  MoveC 456 to (-171.94, 224.64, -10) mm, rotated rx 180 ry 0 rz 0.01 deg; joints [37.11, -45.165, 102.078, -138.154, 64.775, 160.021] to (-186.27, 223.92, -10) mm, rotated rx 180 ry 0 rz 0.01 deg; joints [36.765, -44.661, 101.03, -138.337, 64.242, 159.776]
  MoveL 457 to (-214.9, 224.22, -10) mm, rotated rx -180 ry 0 rz 0.01 deg; joints [36.141, -43.585, 98.793, -138.602, 63.141, 159.21]
  MoveC 458 to (-228.22, 225.49, -10) mm, rotated rx -180 ry 0 rz 0.01 deg; joints [35.891, -43.043, 97.666, -138.663, 62.606, 158.897] to (-241.07, 229.24, -10) mm, rotated rx -180 ry 0 rz 0.01 deg; joints [35.728, -42.444, 96.418, -138.608, 62.056, 158.493]
  MoveC 459 to (-253.06, 235.13, -10) mm, rotated rx -180 ry 0 rz 0.01 deg; joints [35.648, -41.812, 95.099, -138.448, 61.51, 158.018] to (-264.01, 242.79, -10) mm, rotated rx 180 ry 0 rz 0.01 deg; joints [35.642, -41.163, 93.745, -138.197, 60.981, 157.485]
  MoveC 460 to (-273.96, 253.08, -10) mm, rotated rx 180 ry 0 rz 0.01 deg; joints [35.733, -40.471, 92.297, -137.818, 60.457, 156.859] to (-281.3, 265.37, -10) mm, rotated rx -180 ry 0 rz 0.01 deg; joints [35.933, -39.816, 90.927, -137.333, 60.013, 156.197]
  MoveC 461 to (-284.47, 273.38, -10) mm, rotated rx -180 ry 0 rz 0.01 deg; joints [36.095, -39.451, 90.161, -137.006, 59.789, 155.796] to (-286.87, 281.66, -10) mm, rotated rx 180 ry 0 rz 0.01 deg; joints [36.278, -39.106, 89.437, -136.663, 59.592, 155.397]
  MoveC 462 to (-286.56, 286.16, -10) mm, rotated rx -180 ry 0 rz 0.01 deg; joints [36.411, -38.984, 89.179, -136.47, 59.552, 155.217] to (-283.74, 289.67, -10) mm, rotated rx 180 ry 0 rz 0.01 deg; joints [36.567, -38.995, 89.198, -136.31, 59.626, 155.138]
  MoveC 463 to (-280.78, 292.97, -10) mm, rotated rx -180 ry 0 rz 0.01 deg; joints [36.721, -39.019, 89.242, -136.159, 59.709, 155.072] to (-279.73, 297.28, -10) mm, rotated rx 180 ry 0 rz 0.01 deg; joints [36.863, -38.932, 89.056, -135.972, 59.701, 154.917]
  MoveC 464 to (-279.69, 299.8, -10) mm, rotated rx 180 ry 0 rz 0.01 deg; joints [36.934, -38.857, 88.897, -135.864, 59.672, 154.812] to (-279.52, 302.32, -10) mm, rotated rx -180 ry 0 rz 0.01 deg; joints [37.007, -38.787, 88.749, -135.756, 59.649, 154.71]
  MoveC 465 to (-280.39, 304.88, -10) mm, rotated rx 180 ry 0 rz 0.01 deg; joints [37.06, -38.672, 88.51, -135.651, 59.583, 154.581] to (-282.85, 305.96, -10) mm, rotated rx 180 ry 0 rz 0.01 deg; joints [37.038, -38.536, 88.227, -135.613, 59.469, 154.473]
  MoveL 466 to (-366.69, 305.96, -10) mm, rotated rx 180 ry 0 rz 0.01 deg; joints [35.359, -34.828, 80.603, -135.633, 55.88, 152.188]
  MoveC 467 to (-369.42, 304.83, -10) mm, rotated rx 180 ry 0 rz 0.01 deg; joints [35.276, -34.736, 80.417, -135.676, 55.772, 152.159] to (-370.55, 302.11, -10) mm, rotated rx -180 ry 0 rz 0.01 deg; joints [35.181, -34.772, 80.494, -135.797, 55.755, 152.251]
  MoveL 468 to (-370.54, 98.69, -10) mm, rotated rx 180 ry 0 rz 0.01 deg; joints [29.276, -40.424, 92.448, -144.823, 58.123, 160.617]
  MoveC 469 to (-369.42, 95.8, -10) mm, rotated rx 180 ry 0 rz 0.01 deg; joints [29.206, -40.54, 92.694, -144.946, 58.204, 160.746] to (-366.65, 94.41, -10) mm, rotated rx -180 ry 0 rz 0.01 deg; joints [29.211, -40.693, 93.013, -145, 58.342, 160.855]
  MoveC 470 to (-361.84, 93.97, -10) mm, rotated rx -180 ry 0 rz 0.01 deg; joints [29.281, -40.911, 93.465, -145.005, 58.558, 160.971] to (-357.03, 93.56, -10) mm, rotated rx 180 ry 0 rz 0.01 deg; joints [29.353, -41.128, 93.915, -145.008, 58.774, 161.086]
  MoveC 471 to (-352.24, 92.78, -10) mm, rotated rx 180 ry 0 rz 0.01 deg; joints [29.412, -41.351, 94.377, -145.026, 58.991, 161.212] to (-347.65, 91.24, -10) mm, rotated rx -180 ry 0 rz 0.01 deg; joints [29.445, -41.582, 94.859, -145.075, 59.207, 161.36]
  MoveC 472 to (-337.46, 86.07, -10) mm, rotated rx 180 ry 0 rz 0.01 deg; joints [29.463, -42.13, 96.004, -145.257, 59.704, 161.746] to (-328.09, 79.55, -10) mm, rotated rx 180 ry 0 rz 0.01 deg; joints [29.425, -42.669, 97.134, -145.493, 60.177, 162.156]
  MoveC 473 to (-319.86, 71.59, -10) mm, rotated rx 180 ry 0 rz 0.01 deg; joints [29.318, -43.186, 98.222, -145.792, 60.614, 162.585] to (-313.25, 62.25, -10) mm, rotated rx 180 ry 0 rz 0.01 deg; joints [29.137, -43.662, 99.228, -146.155, 60.996, 163.023]
  MoveL 474 to (-295.27, 31.05, -10) mm, rotated rx -180 ry 0 rz 0.01 deg; joints [28.438, -45.048, 102.174, -147.375, 62.088, 164.363]
  MoveC 475 to (-292.31, 25.1, -10) mm, rotated rx 180 ry 0 rz 0.01 deg; joints [28.294, -45.288, 102.686, -147.609, 62.275, 164.603] to (-290.1, 18.82, -10) mm, rotated rx -180 ry 0 rz 0.01 deg; joints [28.123, -45.503, 103.148, -147.862, 62.435, 164.839]
  MoveC 476 to (-288.58, 12.36, -10) mm, rotated rx -180 ry 0 rz 0.01 deg; joints [27.933, -45.694, 103.558, -148.128, 62.567, 165.067] to (-287.65, 5.78, -10) mm, rotated rx -180 ry 0 rz 0.01 deg; joints [27.728, -45.861, 103.921, -148.404, 62.676, 165.287]
  MoveC 477 to (-286.3, 3.07, -10) mm, rotated rx 180 ry 0 rz 0.01 deg; joints [27.66, -45.968, 104.149, -148.51, 62.761, 165.393] to (-283.47, 1.97, -10) mm, rotated rx 180 ry 0 rz 0.01 deg; joints [27.673, -46.101, 104.429, -148.535, 62.89, 165.473]
  MoveL 478 to (-110.06, 1.97, -10) mm, rotated rx 180 ry 0 rz 0.01 deg; joints [31.113, -52.422, 117.77, -146.55, 69.684, 168.087]
  MoveC 479 to (-107.23, 3.06, -10) mm, rotated rx -180 ry 0 rz 0.01 deg; joints [31.215, -52.496, 117.927, -146.461, 69.776, 168.098] to (-105.84, 5.75, -10) mm, rotated rx -180 ry 0 rz 0.01 deg; joints [31.345, -52.491, 117.909, -146.324, 69.796, 168.043]
  MoveC 480 to (-104.8, 12.53, -10) mm, rotated rx -180 ry 0 rz 0.01 deg; joints [31.615, -52.393, 117.685, -146.018, 69.754, 167.869] to (-103.19, 19.2, -10) mm, rotated rx -180 ry 0 rz 0.01 deg; joints [31.892, -52.315, 117.505, -145.709, 69.734, 167.705]
  MoveC 481 to (-100.9, 25.67, -10) mm, rotated rx 180 ry 0 rz 0.01 deg; joints [32.178, -52.262, 117.379, -145.399, 69.742, 167.556] to (-97.83, 31.82, -10) mm, rotated rx -180 ry 0 rz 0.01 deg; joints [32.468, -52.241, 117.321, -145.09, 69.781, 167.426]
  MoveL 482 to (-79.89, 62.85, -10) mm, rotated rx -180 ry 0 rz 0.01 deg; joints [33.989, -52.192, 117.153, -143.496, 70.059, 166.797]
  MoveC 483 to (-73.14, 72.29, -10) mm, rotated rx -180 ry 0 rz 0.01 deg; joints [34.481, -52.212, 117.176, -142.99, 70.187, 166.621] to (-64.7, 80.26, -10) mm, rotated rx -180 ry 0 rz 0.01 deg; joints [34.964, -52.315, 117.38, -142.516, 70.39, 166.513]
  MoveC 484 to (-55.07, 86.69, -10) mm, rotated rx -180 ry 0 rz 0.01 deg; joints [35.424, -52.487, 117.731, -142.083, 70.651, 166.468] to (-44.63, 91.7, -10) mm, rotated rx -180 ry 0 rz 0.01 deg; joints [35.858, -52.711, 118.2, -141.692, 70.955, 166.477]
  MoveC 485 to (-40.32, 93.04, -10) mm, rotated rx 180 ry 0 rz 0.01 deg; joints [36.014, -52.82, 118.428, -141.559, 71.088, 166.502] to (-35.85, 93.69, -10) mm, rotated rx -180 ry 0 rz 0.01 deg; joints [36.15, -52.947, 118.699, -141.45, 71.235, 166.55]
  MoveC 486 to (-31.35, 94.03, -10) mm, rotated rx 180 ry 0 rz 0.01 deg; joints [36.276, -53.082, 118.985, -141.353, 71.386, 166.607] to (-26.86, 94.42, -10) mm, rotated rx -180 ry 0 rz 0.01 deg; joints [36.404, -53.215, 119.269, -141.254, 71.536, 166.663]
  MoveC 487 to (-24.09, 95.8, -10) mm, rotated rx 180 ry 0 rz 0.01 deg; joints [36.524, -53.271, 119.387, -141.145, 71.614, 166.664] to (-22.97, 98.68, -10) mm, rotated rx 180 ry 0 rz 0.01 deg; joints [36.653, -53.242, 119.318, -141.005, 71.617, 166.595]
  MoveL 488 to (-22.97, 302.11, -10) mm, rotated rx -180 ry 0 rz 0.01 deg; joints [43.096, -48.06, 108.004, -133, 69.13, 159.892]
  MoveC 489 to (-24.1, 304.84, -10) mm, rotated rx 180 ry 0 rz 0.01 deg; joints [43.143, -47.946, 107.762, -132.917, 69.06, 159.773] to (-26.83, 305.97, -10) mm, rotated rx -180 ry 0 rz 0.01 deg; joints [43.103, -47.828, 107.512, -132.92, 68.955, 159.685]
  MoveL 490 to (-110.7, 305.97, -10) mm, rotated rx 180 ry 0 rz 0.01 deg; joints [40.945, -45.062, 101.736, -134.176, 66.057, 158.173]
  MoveC 491 to (-113.15, 304.87, -10) mm, rotated rx 180 ry 0 rz 0.01 deg; joints [40.853, -45.009, 101.629, -134.25, 65.983, 158.169] to (-113.97, 302.32, -10) mm, rotated rx -180 ry 0 rz 0.01 deg; joints [40.761, -45.055, 101.728, -134.361, 65.984, 158.249]
  MoveC 492 to (-113.72, 293.56, -10) mm, rotated rx -180 ry 0 rz 0.01 deg; joints [40.516, -45.317, 102.286, -134.701, 66.096, 158.583] to (-114.89, 284.87, -10) mm, rotated rx -180 ry 0 rz 0.01 deg; joints [40.237, -45.525, 102.732, -135.058, 66.157, 158.885]
  MoveC 493 to (-117.34, 276.46, -10) mm, rotated rx 180 ry 0 rz 0.01 deg; joints [39.933, -45.678, 103.064, -135.421, 66.168, 159.151] to (-120.94, 268.47, -10) mm, rotated rx 180 ry 0 rz 0.01 deg; joints [39.612, -45.777, 103.284, -135.783, 66.133, 159.377]
  MoveC 494 to (-124.45, 262.63, -10) mm, rotated rx -180 ry 0 rz 0.01 deg; joints [39.355, -45.818, 103.378, -136.06, 66.076, 159.526] to (-128.5, 257.15, -10) mm, rotated rx 180 ry 0 rz 0.01 deg; joints [39.096, -45.828, 103.408, -136.329, 65.994, 159.651]
  MoveC 495 to (-133.13, 252.15, -10) mm, rotated rx -180 ry 0 rz 0.01 deg; joints [38.837, -45.804, 103.366, -136.587, 65.885, 159.747] to (-138.35, 247.76, -10) mm, rotated rx 180 ry 0 rz 0.01 deg; joints [38.582, -45.741, 103.242, -136.828, 65.747, 159.811]
  MoveC 496 to (-143.45, 244.23, -10) mm, rotated rx -180 ry 0 rz 0.01 deg; joints [38.357, -45.657, 103.072, -137.032, 65.601, 159.844] to (-148.78, 241.05, -10) mm, rotated rx 180 ry 0 rz 0.01 deg; joints [38.137, -45.555, 102.864, -137.224, 65.443, 159.86]
  MoveC 497 to (-154.39, 238.38, -10) mm, rotated rx 180 ry 0 rz 0.01 deg; joints [37.926, -45.427, 102.603, -137.398, 65.267, 159.853] to (-160.28, 236.41, -10) mm, rotated rx 180 ry 0 rz 0.01 deg; joints [37.731, -45.27, 102.278, -137.546, 65.072, 159.814]
  MoveC 498 to (-173.77, 233.82, -10) mm, rotated rx 180 ry 0 rz 0.01 deg; joints [37.343, -44.853, 101.413, -137.802, 64.598, 159.654] to (-187.5, 233.2, -10) mm, rotated rx -180 ry 0 rz 0.01 deg; joints [37.015, -44.367, 100.404, -137.971, 64.087, 159.415]
  MoveL 499 to (-214.9, 233.58, -10) mm, rotated rx -180 ry 0 rz 0.01 deg; joints [36.419, -43.332, 98.253, -138.216, 63.032, 158.863]
  MoveC 500 to (-226.62, 234.71, -10) mm, rotated rx 180 ry 0 rz 0.01 deg; joints [36.198, -42.854, 97.259, -138.269, 62.562, 158.584] to (-237.91, 238.06, -10) mm, rotated rx 180 ry 0 rz 0.01 deg; joints [36.054, -42.325, 96.158, -138.219, 62.079, 158.225]
  MoveC 501 to (-248.45, 243.28, -10) mm, rotated rx 180 ry 0 rz 0.01 deg; joints [35.983, -41.768, 94.996, -138.077, 61.6, 157.803] to (-258.07, 250.02, -10) mm, rotated rx -180 ry 0 rz 0.01 deg; joints [35.976, -41.198, 93.805, -137.857, 61.136, 157.333]
  MoveC 502 to (-265.05, 256.9, -10) mm, rotated rx 180 ry 0 rz 0.01 deg; joints [36.028, -40.723, 92.812, -137.61, 60.774, 156.908] to (-270.66, 264.93, -10) mm, rotated rx -180 ry 0 rz 0.01 deg; joints [36.141, -40.265, 91.854, -137.302, 60.453, 156.46]
  MoveC 503 to (-274.9, 273.74, -10) mm, rotated rx -180 ry 0 rz 0.01 deg; joints [36.303, -39.835, 90.953, -136.95, 60.177, 156.006] to (-277.86, 283.05, -10) mm, rotated rx -180 ry 0 rz 0.01 deg; joints [36.504, -39.438, 90.12, -136.569, 59.946, 155.555]
  MoveC 504 to (-278.84, 287.81, -10) mm, rotated rx -180 ry 0 rz 0.01 deg; joints [36.617, -39.255, 89.736, -136.371, 59.849, 155.334] to (-279.48, 292.62, -10) mm, rotated rx -180 ry 0 rz 0.01 deg; joints [36.738, -39.084, 89.375, -136.169, 59.766, 155.118]
  MoveC 505 to (-279.66, 294.95, -10) mm, rotated rx -180 ry 0 rz 0.01 deg; joints [36.799, -39.006, 89.212, -136.071, 59.731, 155.017] to (-279.73, 297.28, -10) mm, rotated rx 180 ry 0 rz 0.01 deg; joints [36.863, -38.932, 89.056, -135.972, 59.701, 154.917]
  MoveC 506 to (-278.37, 301.48, -10) mm, rotated rx 180 ry 0 rz 0.01 deg; joints [37.008, -38.86, 88.902, -135.788, 59.706, 154.774] to (-274.78, 304.03, -10) mm, rotated rx 180 ry 0 rz 0.01 deg; joints [37.154, -38.931, 89.044, -135.666, 59.823, 154.754]
  MoveC 507 to (-271.13, 306.39, -10) mm, rotated rx 180 ry 0 rz 0.01 deg; joints [37.296, -39.01, 89.203, -135.552, 59.944, 154.743] to (-269.26, 310.32, -10) mm, rotated rx 180 ry 0 rz 0.01 deg; joints [37.444, -38.966, 89.107, -135.378, 59.973, 154.623]
  MoveL 508 to (-269.1, 311.3, -10) mm, rotated rx 180 ry 0 rz 0.01 deg; joints [37.474, -38.942, 89.057, -135.336, 59.968, 154.585]
  MoveC 509 to (-269.84, 313.86, -10) mm, rotated rx 180 ry 0 rz 0.01 deg; joints [37.53, -38.832, 88.827, -135.23, 59.907, 154.458] to (-272.26, 314.98, -10) mm, rotated rx -180 ry 0 rz 0.01 deg; joints [37.509, -38.697, 88.547, -135.192, 59.795, 154.351]
  MoveL 510 to (-375.71, 314.98, -10) mm, rotated rx -180 ry 0 rz 0.01 deg; joints [35.43, -34.104, 79.107, -135.188, 55.364, 151.488]
  MoveC 511 to (-378.44, 313.85, -10) mm, rotated rx -180 ry 0 rz 0.01 deg; joints [35.347, -34.012, 78.918, -135.228, 55.255, 151.456] to (-379.56, 311.12, -10) mm, rotated rx -180 ry 0 rz 0.01 deg; joints [35.253, -34.048, 78.997, -135.349, 55.238, 151.551]
  MoveL 512 to (-379.56, 88.8, -10) mm, rotated rx -180 ry 0 rz 0.01 deg; joints [28.815, -40.261, 92.128, -145.276, 57.831, 160.785]
  MoveC 513 to (-378.48, 86.36, -10) mm, rotated rx 180 ry 0 rz 0.01 deg; joints [28.758, -40.365, 92.347, -145.38, 57.906, 160.897] to (-375.96, 85.52, -10) mm, rotated rx -180 ry 0 rz 0.01 deg; joints [28.774, -40.495, 92.618, -145.412, 58.028, 160.981]
  MoveC 514 to (-365.44, 85.57, -10) mm, rotated rx -180 ry 0 rz 0.01 deg; joints [28.957, -40.951, 93.561, -145.382, 58.492, 161.199] to (-355.08, 83.79, -10) mm, rotated rx -180 ry 0 rz 0.01 deg; joints [29.081, -41.437, 94.571, -145.426, 58.966, 161.474]
  MoveC 515 to (-345.19, 80.2, -10) mm, rotated rx 180 ry 0 rz 0.01 deg; joints [29.142, -41.938, 95.617, -145.543, 59.435, 161.799] to (-336.12, 74.87, -10) mm, rotated rx -180 ry 0 rz 0.01 deg; joints [29.133, -42.439, 96.666, -145.734, 59.884, 162.162]
  MoveC 516 to (-332.09, 71.59, -10) mm, rotated rx -180 ry 0 rz 0.01 deg; joints [29.1, -42.681, 97.173, -145.856, 60.093, 162.353] to (-328.5, 67.83, -10) mm, rotated rx -180 ry 0 rz 0.01 deg; joints [29.043, -42.913, 97.662, -146, 60.287, 162.55]
  MoveC 517 to (-325.25, 63.78, -10) mm, rotated rx -180 ry 0 rz 0.01 deg; joints [28.971, -43.137, 98.133, -146.157, 60.47, 162.749] to (-322.21, 59.57, -10) mm, rotated rx 180 ry 0 rz 0.01 deg; joints [28.89, -43.354, 98.592, -146.322, 60.645, 162.947]
  MoveL 518 to (-303.09, 26.55, -10) mm, rotated rx -180 ry 0 rz 0.01 deg; joints [28.149, -44.829, 101.724, -147.622, 61.809, 164.373]
  MoveC 519 to (-300.41, 21.16, -10) mm, rotated rx 180 ry 0 rz 0.01 deg; joints [28.018, -45.046, 102.188, -147.836, 61.979, 164.591] to (-298.41, 15.48, -10) mm, rotated rx -180 ry 0 rz 0.01 deg; joints [27.864, -45.241, 102.605, -148.065, 62.124, 164.805]
  MoveC 520 to (-297.06, 9.62, -10) mm, rotated rx -180 ry 0 rz 0.01 deg; joints [27.691, -45.412, 102.974, -148.308, 62.242, 165.012] to (-296.31, 3.65, -10) mm, rotated rx 180 ry 0 rz 0.01 deg; joints [27.503, -45.56, 103.295, -148.559, 62.337, 165.211]
  MoveC 521 to (-296.27, 1.93, -10) mm, rotated rx 180 ry 0 rz 0.01 deg; joints [27.445, -45.596, 103.374, -148.633, 62.357, 165.265] to (-296.38, 0.21, -10) mm, rotated rx 180 ry 0 rz 0.01 deg; joints [27.385, -45.626, 103.439, -148.708, 62.371, 165.317]
  MoveC 522 to (-296.54, -1.51, -10) mm, rotated rx -180 ry 0 rz 0.01 deg; joints [27.324, -45.653, 103.499, -148.783, 62.382, 165.368] to (-296.65, -3.23, -10) mm, rotated rx 180 ry 0 rz 0.01 deg; joints [27.264, -45.682, 103.563, -148.858, 62.396, 165.419]
  MoveC 523 to (-295.65, -5.92, -10) mm, rotated rx -180 ry 0 rz 0.01 deg; joints [27.19, -45.774, 103.761, -148.966, 62.466, 165.518] to (-293.02, -7.04, -10) mm, rotated rx 180 ry 0 rz 0.01 deg; joints [27.198, -45.9, 104.027, -148.995, 62.588, 165.596]
  MoveL 524 to (-100.49, -7.04, -10) mm, rotated rx 180 ry 0 rz 0.01 deg; joints [30.994, -52.918, 118.849, -146.791, 70.144, 168.472]
  MoveC 525 to (-97.86, -5.92, -10) mm, rotated rx 180 ry 0 rz 0.01 deg; joints [31.094, -52.985, 118.989, -146.702, 70.228, 168.479] to (-96.86, -3.23, -10) mm, rotated rx 180 ry 0 rz 0.01 deg; joints [31.215, -52.967, 118.945, -146.571, 70.233, 168.42]
  MoveC 526 to (-97.01, 0.21, -10) mm, rotated rx -180 ry 0 rz 0.01 deg; joints [31.339, -52.895, 118.784, -146.425, 70.187, 168.323] to (-97.13, 3.65, -10) mm, rotated rx 180 ry 0 rz 0.01 deg; joints [31.462, -52.824, 118.625, -146.28, 70.141, 168.226]
  MoveC 527 to (-96.99, 7.1, -10) mm, rotated rx 180 ry 0 rz 0.01 deg; joints [31.592, -52.762, 118.484, -146.13, 70.106, 168.133] to (-96.32, 10.49, -10) mm, rotated rx -180 ry 0 rz 0.01 deg; joints [31.731, -52.717, 118.383, -145.974, 70.09, 168.048]
  MoveC 528 to (-95.07, 14.81, -10) mm, rotated rx -180 ry 0 rz 0.01 deg; joints [31.916, -52.674, 118.28, -145.77, 70.084, 167.946] to (-93.71, 19.1, -10) mm, rotated rx 180 ry 0 rz 0.01 deg; joints [32.103, -52.634, 118.187, -145.566, 70.083, 167.845]
  MoveC 529 to (-92.08, 23.3, -10) mm, rotated rx -180 ry 0 rz 0.01 deg; joints [32.293, -52.605, 118.115, -145.361, 70.093, 167.751] to (-90.02, 27.3, -10) mm, rotated rx 180 ry 0 rz 0.01 deg; joints [32.485, -52.593, 118.081, -145.159, 70.12, 167.668]
  MoveL 530 to (-72.09, 58.34, -10) mm, rotated rx 180 ry 0 rz 0.01 deg; joints [34.015, -52.544, 117.912, -143.556, 70.393, 167.044]
  MoveC 531 to (-66.2, 66.54, -10) mm, rotated rx -180 ry 0 rz 0.01 deg; joints [34.447, -52.563, 117.934, -143.113, 70.504, 166.894] to (-58.81, 73.43, -10) mm, rotated rx -180 ry 0 rz 0.01 deg; joints [34.869, -52.655, 118.116, -142.699, 70.681, 166.803]
  MoveC 532 to (-50.41, 78.97, -10) mm, rotated rx -180 ry 0 rz 0.01 deg; joints [35.271, -52.806, 118.427, -142.321, 70.909, 166.766] to (-41.32, 83.31, -10) mm, rotated rx -180 ry 0 rz 0.01 deg; joints [35.649, -53.002, 118.837, -141.979, 71.173, 166.774]
  MoveC 533 to (-35.54, 85.06, -10) mm, rotated rx 180 ry 0 rz 0.01 deg; joints [35.856, -53.147, 119.144, -141.801, 71.353, 166.81] to (-29.56, 85.81, -10) mm, rotated rx 180 ry 0 rz 0.01 deg; joints [36.034, -53.32, 119.511, -141.66, 71.55, 166.877]
  MoveC 534 to (-23.55, 85.87, -10) mm, rotated rx -180 ry 0 rz 0.01 deg; joints [36.19, -53.508, 119.913, -141.545, 71.757, 166.965] to (-17.55, 85.52, -10) mm, rotated rx 180 ry 0 rz 0.01 deg; joints [36.333, -53.704, 120.332, -141.445, 71.967, 167.065]
  MoveC 535 to (-15.02, 86.36, -10) mm, rotated rx 180 ry 0 rz 0.01 deg; joints [36.428, -53.764, 120.459, -141.362, 72.043, 167.078] to (-13.95, 88.8, -10) mm, rotated rx 180 ry 0 rz 0.01 deg; joints [36.541, -53.743, 120.411, -141.24, 72.049, 167.022]
  MoveL 536 to (-13.96, 311.13, -10) mm, rotated rx -180 ry 0 rz 0.01 deg; joints [43.598, -48.082, 108.038, -132.504, 69.322, 159.718]
  MoveC 537 to (-15.09, 313.86, -10) mm, rotated rx 180 ry 0 rz 0.01 deg; joints [43.645, -47.968, 107.794, -132.421, 69.252, 159.599] to (-17.81, 314.99, -10) mm, rotated rx 180 ry 0 rz 0.01 deg; joints [43.603, -47.85, 107.545, -132.426, 69.148, 159.511]
  MoveL 538 to (-121.25, 314.98, -10) mm, rotated rx 180 ry 0 rz 0.01 deg; joints [40.941, -44.432, 100.412, -133.956, 65.573, 157.628]
  MoveC 539 to (-123.66, 313.88, -10) mm, rotated rx 180 ry 0 rz 0.01 deg; joints [40.851, -44.38, 100.307, -134.028, 65.499, 157.624] to (-124.39, 311.33, -10) mm, rotated rx 180 ry 0 rz 0.01 deg; joints [40.761, -44.429, 100.413, -134.137, 65.503, 157.707]
  MoveC 540 to (-123.61, 306.3, -10) mm, rotated rx 180 ry 0 rz 0.01 deg; joints [40.638, -44.604, 100.784, -134.325, 65.59, 157.915] to (-122.74, 301.29, -10) mm, rotated rx -180 ry 0 rz 0.01 deg; joints [40.516, -44.781, 101.158, -134.512, 65.681, 158.122]
  MoveC 541 to (-122.36, 296.18, -10) mm, rotated rx -180 ry 0 rz 0.01 deg; joints [40.38, -44.942, 101.501, -134.708, 65.755, 158.322] to (-123.02, 291.11, -10) mm, rotated rx -180 ry 0 rz 0.01 deg; joints [40.218, -45.065, 101.765, -134.916, 65.791, 158.5]
  MoveC 542 to (-124.39, 285.57, -10) mm, rotated rx 180 ry 0 rz 0.01 deg; joints [40.025, -45.175, 102.004, -135.152, 65.807, 158.681] to (-125.85, 280.05, -10) mm, rotated rx -180 ry 0 rz 0.01 deg; joints [39.83, -45.281, 102.233, -135.388, 65.819, 158.859]
  MoveC 543 to (-127.85, 274.68, -10) mm, rotated rx 180 ry 0 rz 0.01 deg; joints [39.626, -45.363, 102.412, -135.626, 65.81, 159.021] to (-130.75, 269.73, -10) mm, rotated rx -180 ry 0 rz 0.01 deg; joints [39.412, -45.4, 102.497, -135.858, 65.764, 159.149]
  MoveC 544 to (-137.55, 261.35, -10) mm, rotated rx 180 ry 0 rz 0.01 deg; joints [39.003, -45.396, 102.5, -136.276, 65.616, 159.331] to (-145.33, 253.87, -10) mm, rotated rx -180 ry 0 rz 0.01 deg; joints [38.598, -45.327, 102.37, -136.669, 65.419, 159.459]
  MoveC 545 to (-154.45, 247.98, -10) mm, rotated rx 180 ry 0 rz 0.01 deg; joints [38.21, -45.164, 102.04, -137.013, 65.152, 159.503] to (-164.79, 244.63, -10) mm, rotated rx -180 ry 0 rz 0.01 deg; joints [37.871, -44.885, 101.463, -137.266, 64.808, 159.43]
  MoveL 546 to (-172.31, 243.24, -10) mm, rotated rx -180 ry 0 rz 0.01 deg; joints [37.657, -44.65, 100.977, -137.404, 64.543, 159.338]
  MoveC 547 to (-175.81, 242.75, -10) mm, rotated rx 180 ry 0 rz 0.01 deg; joints [37.563, -44.536, 100.74, -137.462, 64.417, 159.289] to (-179.35, 242.59, -10) mm, rotated rx -180 ry 0 rz 0.01 deg; joints [37.477, -44.411, 100.481, -137.506, 64.286, 159.227]
  MoveL 548 to (-214.9, 242.6, -10) mm, rotated rx 180 ry 0 rz 0.01 deg; joints [36.685, -43.085, 97.726, -137.846, 62.926, 158.525]
  MoveC 549 to (-225.08, 243.6, -10) mm, rotated rx 180 ry 0 rz 0.01 deg; joints [36.492, -42.669, 96.861, -137.89, 62.518, 158.28] to (-234.87, 246.55, -10) mm, rotated rx -180 ry 0 rz 0.01 deg; joints [36.367, -42.208, 95.903, -137.844, 62.099, 157.964]
  MoveC 550 to (-244, 251.12, -10) mm, rotated rx 180 ry 0 rz 0.01 deg; joints [36.305, -41.724, 94.892, -137.72, 61.685, 157.594] to (-252.35, 256.99, -10) mm, rotated rx -180 ry 0 rz 0.01 deg; joints [36.298, -41.228, 93.857, -137.53, 61.283, 157.184]
  MoveC 551 to (-258.28, 262.86, -10) mm, rotated rx -180 ry 0 rz 0.01 deg; joints [36.341, -40.824, 93.013, -137.321, 60.977, 156.822] to (-263.02, 269.72, -10) mm, rotated rx -180 ry 0 rz 0.01 deg; joints [36.437, -40.435, 92.199, -137.06, 60.706, 156.442]
  MoveC 552 to (-266.59, 277.24, -10) mm, rotated rx 180 ry 0 rz 0.01 deg; joints [36.576, -40.071, 91.435, -136.762, 60.473, 156.056] to (-269.1, 285.18, -10) mm, rotated rx -180 ry 0 rz 0.01 deg; joints [36.747, -39.734, 90.728, -136.44, 60.278, 155.674]
  MoveC 553 to (-269.97, 289.19, -10) mm, rotated rx 180 ry 0 rz 0.01 deg; joints [36.841, -39.579, 90.401, -136.274, 60.195, 155.488] to (-270.64, 293.25, -10) mm, rotated rx 180 ry 0 rz 0.01 deg; joints [36.941, -39.429, 90.087, -136.106, 60.119, 155.304]
  MoveC 554 to (-270.98, 297.35, -10) mm, rotated rx 180 ry 0 rz 0.01 deg; joints [37.048, -39.291, 89.797, -135.934, 60.057, 155.126] to (-270.86, 301.47, -10) mm, rotated rx 180 ry 0 rz 0.01 deg; joints [37.165, -39.171, 89.543, -135.759, 60.013, 154.957]
  MoveC 555 to (-270.55, 303.95, -10) mm, rotated rx 180 ry 0 rz 0.01 deg; joints [37.24, -39.108, 89.41, -135.653, 59.996, 154.86] to (-270.06, 306.4, -10) mm, rotated rx -180 ry 0 rz 0.01 deg; joints [37.319, -39.054, 89.293, -135.547, 59.987, 154.769]
  MoveC 556 to (-269.63, 308.35, -10) mm, rotated rx -180 ry 0 rz 0.01 deg; joints [37.382, -39.011, 89.204, -135.463, 59.981, 154.697] to (-269.26, 310.32, -10) mm, rotated rx 180 ry 0 rz 0.01 deg; joints [37.444, -38.966, 89.107, -135.378, 59.973, 154.623]
  MoveC 557 to (-267.76, 313.87, -10) mm, rotated rx 180 ry 0 rz 0.01 deg; joints [37.574, -38.918, 89.003, -135.221, 59.992, 154.509] to (-264.83, 316.39, -10) mm, rotated rx -180 ry 0 rz 0.01 deg; joints [37.705, -38.96, 89.087, -135.103, 60.081, 154.474]
  MoveC 558 to (-262.85, 320.74, -10) mm, rotated rx -180 ry 0 rz 0.01 deg; joints [37.867, -38.906, 88.969, -134.911, 60.109, 154.337] to (-266.61, 323.69, -10) mm, rotated rx -180 ry 0 rz 0.01 deg; joints [37.868, -38.659, 88.455, -134.801, 59.921, 154.119]
  MoveL 559 to (-384.43, 323.69, -10) mm, rotated rx -180 ry 0 rz 0.01 deg; joints [35.497, -33.392, 77.634, -134.742, 54.861, 150.791]
  MoveC 560 to (-387.15, 322.56, -10) mm, rotated rx -180 ry 0 rz 0.01 deg; joints [35.415, -33.297, 77.442, -134.78, 54.751, 150.757] to (-388.28, 319.84, -10) mm, rotated rx -180 ry 0 rz 0.01 deg; joints [35.321, -33.335, 77.522, -134.9, 54.733, 150.853]
  MoveL 561 to (-388.27, 77.07, -10) mm, rotated rx -180 ry 0 rz 0.01 deg; joints [28.303, -40.148, 91.916, -145.807, 57.57, 161.027]
  MoveC 562 to (-387.15, 74.83, -10) mm, rotated rx -180 ry 0 rz 0.01 deg; joints [28.252, -40.249, 92.128, -145.903, 57.645, 161.132] to (-384.69, 74.39, -10) mm, rotated rx 180 ry 0 rz 0.01 deg; joints [28.28, -40.368, 92.374, -145.918, 57.76, 161.2]
  MoveC 563 to (-381.03, 75.49, -10) mm, rotated rx 180 ry 0 rz 0.01 deg; joints [28.376, -40.504, 92.653, -145.862, 57.911, 161.237] to (-377.39, 76.6, -10) mm, rotated rx -180 ry 0 rz 0.01 deg; joints [28.472, -40.638, 92.929, -145.805, 58.062, 161.273]
  MoveC 564 to (-373.63, 77.36, -10) mm, rotated rx -180 ry 0 rz 0.01 deg; joints [28.56, -40.784, 93.23, -145.762, 58.22, 161.324] to (-369.8, 77.38, -10) mm, rotated rx -180 ry 0 rz 0.01 deg; joints [28.626, -40.95, 93.574, -145.751, 58.389, 161.402]
  MoveC 565 to (-360.78, 76.03, -10) mm, rotated rx 180 ry 0 rz 0.01 deg; joints [28.738, -41.37, 94.445, -145.782, 58.801, 161.634] to (-351.95, 73.74, -10) mm, rotated rx -180 ry 0 rz 0.01 deg; joints [28.819, -41.798, 95.338, -145.85, 59.212, 161.892]
  MoveC 566 to (-343.66, 69.76, -10) mm, rotated rx 180 ry 0 rz 0.01 deg; joints [28.838, -42.238, 96.256, -145.988, 59.615, 162.193] to (-336.77, 63.67, -10) mm, rotated rx -180 ry 0 rz 0.01 deg; joints [28.764, -42.661, 97.146, -146.22, 59.978, 162.535]
  MoveC 567 to (-334.62, 61.18, -10) mm, rotated rx -180 ry 0 rz 0.01 deg; joints [28.722, -42.805, 97.45, -146.317, 60.097, 162.661] to (-332.45, 58.72, -10) mm, rotated rx -180 ry 0 rz 0.01 deg; joints [28.681, -42.949, 97.753, -146.413, 60.217, 162.785]
  MoveC 568 to (-330.4, 56.16, -10) mm, rotated rx 180 ry 0 rz 0.01 deg; joints [28.635, -43.09, 98.051, -146.513, 60.333, 162.911] to (-328.61, 53.39, -10) mm, rotated rx -180 ry 0 rz 0.01 deg; joints [28.577, -43.224, 98.334, -146.622, 60.439, 163.037]
  MoveL 569 to (-310.64, 22.2, -10) mm, rotated rx -180 ry 0 rz 0.01 deg; joints [27.872, -44.614, 101.284, -147.859, 61.538, 164.383]
  MoveC 570 to (-307.03, 14.06, -10) mm, rotated rx -180 ry 0 rz 0.01 deg; joints [27.664, -44.924, 101.947, -148.185, 61.776, 164.704] to (-305.21, 5.36, -10) mm, rotated rx 180 ry 0 rz 0.01 deg; joints [27.405, -45.172, 102.48, -148.548, 61.946, 165.01]
  MoveC 571 to (-305.03, -3.52, -10) mm, rotated rx 180 ry 0 rz 0.01 deg; joints [27.109, -45.354, 102.877, -148.929, 62.047, 165.291] to (-306.26, -12.31, -10) mm, rotated rx -180 ry 0 rz 0.01 deg; joints [26.79, -45.475, 103.147, -149.316, 62.087, 165.543]
  MoveC 572 to (-305.71, -14.7, -10) mm, rotated rx -180 ry 0 rz 0.01 deg; joints [26.718, -45.543, 103.294, -149.416, 62.135, 165.626] to (-303.5, -15.76, -10) mm, rotated rx 180 ry 0 rz 0.01 deg; joints [26.72, -45.652, 103.524, -149.446, 62.24, 165.694]
  MoveL 573 to (-89.98, -15.76, -10) mm, rotated rx 180 ry 0 rz 0.01 deg; joints [30.904, -53.435, 119.975, -147.002, 70.634, 168.857]
  MoveC 574 to (-87.77, -14.68, -10) mm, rotated rx 180 ry 0 rz 0.01 deg; joints [30.994, -53.488, 120.086, -146.921, 70.703, 168.859] to (-87.24, -12.28, -10) mm, rotated rx 180 ry 0 rz 0.01 deg; joints [31.095, -53.46, 120.021, -146.809, 70.693, 168.802]
  MoveC 575 to (-88.5, -3.69, -10) mm, rotated rx -180 ry 0 rz 0.01 deg; joints [31.386, -53.254, 119.561, -146.459, 70.545, 168.551] to (-88.14, 4.98, -10) mm, rotated rx 180 ry 0 rz 0.01 deg; joints [31.714, -53.098, 119.208, -146.081, 70.455, 168.318]
  MoveC 576 to (-86.31, 13.45, -10) mm, rotated rx -180 ry 0 rz 0.01 deg; joints [32.066, -52.993, 118.964, -145.689, 70.42, 168.11] to (-83.21, 21.54, -10) mm, rotated rx 180 ry 0 rz 0.01 deg; joints [32.433, -52.935, 118.822, -145.294, 70.436, 167.929]
  MoveL 577 to (-64.54, 53.98, -10) mm, rotated rx 180 ry 0 rz 0.01 deg; joints [34.042, -52.883, 118.643, -143.611, 70.715, 167.282]
  MoveC 578 to (-59.48, 60.99, -10) mm, rotated rx 180 ry 0 rz 0.01 deg; joints [34.413, -52.899, 118.663, -143.23, 70.809, 167.155] to (-53.12, 66.83, -10) mm, rotated rx -180 ry 0 rz 0.01 deg; joints [34.776, -52.98, 118.824, -142.875, 70.963, 167.08]
  MoveC 579 to (-45.89, 71.52, -10) mm, rotated rx 180 ry 0 rz 0.01 deg; joints [35.12, -53.112, 119.095, -142.551, 71.159, 167.051] to (-38.11, 75.21, -10) mm, rotated rx -180 ry 0 rz 0.01 deg; joints [35.445, -53.28, 119.448, -142.257, 71.385, 167.059]
  MoveC 580 to (-33.55, 76.59, -10) mm, rotated rx 180 ry 0 rz 0.01 deg; joints [35.609, -53.395, 119.691, -142.116, 71.527, 167.087] to (-28.83, 77.21, -10) mm, rotated rx 180 ry 0 rz 0.01 deg; joints [35.75, -53.531, 119.98, -142.003, 71.682, 167.139]
  MoveC 581 to (-24.09, 77.33, -10) mm, rotated rx -180 ry 0 rz 0.01 deg; joints [35.875, -53.678, 120.294, -141.909, 71.845, 167.207] to (-19.34, 77.24, -10) mm, rotated rx -180 ry 0 rz 0.01 deg; joints [35.994, -53.828, 120.617, -141.822, 72.009, 167.279]
  MoveC 582 to (-16.62, 76.91, -10) mm, rotated rx 180 ry 0 rz 0.01 deg; joints [36.053, -53.921, 120.815, -141.784, 72.107, 167.329] to (-13.99, 76.14, -10) mm, rotated rx -180 ry 0 rz 0.01 deg; joints [36.093, -54.019, 121.028, -141.765, 72.207, 167.391]
  MoveC 583 to (-11.42, 75.2, -10) mm, rotated rx 180 ry 0 rz 0.01 deg; joints [36.127, -54.119, 121.245, -141.755, 72.306, 167.456] to (-8.82, 74.37, -10) mm, rotated rx 180 ry 0 rz 0.01 deg; joints [36.165, -54.218, 121.459, -141.739, 72.406, 167.518]
  MoveC 584 to (-6.36, 74.8, -10) mm, rotated rx 180 ry 0 rz 0.01 deg; joints [36.244, -54.285, 121.602, -141.672, 72.484, 167.542] to (-5.24, 77.03, -10) mm, rotated rx -180 ry 0 rz 0.01 deg; joints [36.353, -54.271, 121.567, -141.558, 72.494, 167.495]
  MoveL 585 to (-5.24, 319.85, -10) mm, rotated rx 180 ry 0 rz 0.01 deg; joints [44.083, -48.099, 108.06, -132.024, 69.506, 159.548]
  MoveC 586 to (-6.37, 322.57, -10) mm, rotated rx -180 ry 0 rz 0.01 deg; joints [44.129, -47.985, 107.816, -131.942, 69.436, 159.428] to (-9.1, 323.7, -10) mm, rotated rx -180 ry 0 rz 0.01 deg; joints [44.087, -47.867, 107.568, -131.948, 69.333, 159.34]
  MoveL 587 to (-134.69, 323.7, -10) mm, rotated rx -180 ry 0 rz 0.01 deg; joints [40.859, -43.7, 98.879, -133.772, 64.984, 157.028]
  MoveC 588 to (-136.66, 322.58, -10) mm, rotated rx 180 ry 0 rz 0.01 deg; joints [40.78, -43.664, 98.806, -133.839, 64.926, 157.032] to (-136.7, 320.32, -10) mm, rotated rx -180 ry 0 rz 0.01 deg; joints [40.716, -43.73, 98.946, -133.928, 64.951, 157.119]
  MoveC 589 to (-135.51, 318.07, -10) mm, rotated rx 180 ry 0 rz 0.01 deg; joints [40.682, -43.839, 99.176, -134.004, 65.021, 157.23] to (-134.36, 315.81, -10) mm, rotated rx -180 ry 0 rz 0.01 deg; joints [40.646, -43.947, 99.404, -134.08, 65.089, 157.341]
  MoveC 590 to (-133.4, 313.44, -10) mm, rotated rx 180 ry 0 rz 0.01 deg; joints [40.602, -44.051, 99.623, -134.162, 65.152, 157.451] to (-132.83, 310.95, -10) mm, rotated rx -180 ry 0 rz 0.01 deg; joints [40.546, -44.144, 99.821, -134.253, 65.202, 157.558]
  MoveC 591 to (-132.12, 306.52, -10) mm, rotated rx 180 ry 0 rz 0.01 deg; joints [40.438, -44.299, 100.15, -134.42, 65.28, 157.742] to (-131.31, 302.1, -10) mm, rotated rx 180 ry 0 rz 0.01 deg; joints [40.332, -44.457, 100.484, -134.585, 65.361, 157.926]
  MoveC 592 to (-130.93, 297.6, -10) mm, rotated rx -180 ry 0 rz 0.01 deg; joints [40.213, -44.601, 100.79, -134.757, 65.428, 158.105] to (-131.5, 293.12, -10) mm, rotated rx 180 ry 0 rz 0.01 deg; joints [40.071, -44.71, 101.024, -134.941, 65.46, 158.263]
  MoveL 593 to (-133.79, 283.65, -10) mm, rotated rx -180 ry 0 rz 0.01 deg; joints [39.743, -44.901, 101.436, -135.344, 65.489, 158.575]
  MoveC 594 to (-135.4, 279.03, -10) mm, rotated rx -180 ry 0 rz 0.01 deg; joints [39.571, -44.976, 101.599, -135.547, 65.485, 158.717] to (-137.85, 274.79, -10) mm, rotated rx -180 ry 0 rz 0.01 deg; joints [39.389, -45.009, 101.675, -135.745, 65.446, 158.829]
  MoveC 595 to (-143.55, 267.66, -10) mm, rotated rx 180 ry 0 rz 0.01 deg; joints [39.046, -45.008, 101.683, -136.097, 65.321, 158.985] to (-150.01, 261.22, -10) mm, rotated rx 180 ry 0 rz 0.01 deg; joints [38.704, -44.958, 101.589, -136.43, 65.16, 159.101]
  MoveC 596 to (-157.64, 256.08, -10) mm, rotated rx 180 ry 0 rz 0.01 deg; joints [38.375, -44.827, 101.325, -136.724, 64.939, 159.145] to (-166.37, 253.2, -10) mm, rotated rx -180 ry 0 rz 0.01 deg; joints [38.088, -44.593, 100.841, -136.938, 64.648, 159.085]
  MoveC 597 to (-169.6, 252.59, -10) mm, rotated rx -180 ry 0 rz 0.01 deg; joints [37.995, -44.492, 100.634, -136.997, 64.535, 159.046] to (-172.82, 251.96, -10) mm, rotated rx 180 ry 0 rz 0.01 deg; joints [37.903, -44.393, 100.428, -137.058, 64.421, 159.007]
  MoveC 598 to (-176.06, 251.47, -10) mm, rotated rx -180 ry 0 rz 0.01 deg; joints [37.814, -44.288, 100.21, -137.112, 64.305, 158.962] to (-179.35, 251.31, -10) mm, rotated rx 180 ry 0 rz 0.01 deg; joints [37.735, -44.172, 99.97, -137.153, 64.184, 158.905]
  MoveL 599 to (-214.9, 251.31, -10) mm, rotated rx -180 ry 0 rz 0.01 deg; joints [36.94, -42.844, 97.212, -137.488, 62.824, 158.196]
  MoveC 600 to (-223.59, 252.18, -10) mm, rotated rx 180 ry 0 rz 0.01 deg; joints [36.776, -42.487, 96.472, -137.524, 62.476, 157.983] to (-231.94, 254.75, -10) mm, rotated rx 180 ry 0 rz 0.01 deg; joints [36.669, -42.093, 95.65, -137.482, 62.119, 157.71]
  MoveC 601 to (-239.7, 258.7, -10) mm, rotated rx -180 ry 0 rz 0.01 deg; joints [36.616, -41.678, 94.786, -137.375, 61.766, 157.392] to (-246.82, 263.73, -10) mm, rotated rx 180 ry 0 rz 0.01 deg; joints [36.609, -41.255, 93.902, -137.214, 61.425, 157.04]
  MoveC 602 to (-251.74, 268.62, -10) mm, rotated rx 180 ry 0 rz 0.01 deg; joints [36.644, -40.919, 93.201, -137.041, 61.172, 156.739] to (-255.64, 274.35, -10) mm, rotated rx 180 ry 0 rz 0.01 deg; joints [36.725, -40.597, 92.526, -136.824, 60.948, 156.422]
  MoveC 603 to (-258.56, 280.63, -10) mm, rotated rx 180 ry 0 rz 0.01 deg; joints [36.841, -40.296, 91.895, -136.578, 60.757, 156.103] to (-260.63, 287.23, -10) mm, rotated rx 180 ry 0 rz 0.01 deg; joints [36.983, -40.017, 91.31, -136.312, 60.596, 155.787]
  MoveC 604 to (-261.88, 294.87, -10) mm, rotated rx -180 ry 0 rz 0.01 deg; joints [37.171, -39.738, 90.721, -135.996, 60.455, 155.444] to (-261.98, 302.62, -10) mm, rotated rx -180 ry 0 rz 0.01 deg; joints [37.385, -39.499, 90.218, -135.671, 60.359, 155.12]
  MoveC 605 to (-260.82, 310.29, -10) mm, rotated rx 180 ry 0 rz 0.01 deg; joints [37.622, -39.313, 89.822, -135.342, 60.315, 154.828] to (-258.32, 317.64, -10) mm, rotated rx -180 ry 0 rz 0.01 deg; joints [37.878, -39.188, 89.554, -135.022, 60.329, 154.579]
  MoveC 606 to (-257.98, 318.33, -10) mm, rotated rx -180 ry 0 rz 0.01 deg; joints [37.905, -39.18, 89.537, -134.991, 60.334, 154.557] to (-257.6, 318.99, -10) mm, rotated rx -180 ry 0 rz 0.01 deg; joints [37.931, -39.175, 89.526, -134.961, 60.341, 154.539]
  MoveC 607 to (-257.2, 319.65, -10) mm, rotated rx -180 ry 0 rz 0.01 deg; joints [37.958, -39.171, 89.517, -134.932, 60.35, 154.52] to (-256.82, 320.32, -10) mm, rotated rx -180 ry 0 rz 0.01 deg; joints [37.984, -39.166, 89.504, -134.902, 60.357, 154.501]
  MoveC 608 to (-256.87, 322.58, -10) mm, rotated rx -180 ry 0 rz 0.01 deg; joints [38.045, -39.093, 89.353, -134.807, 60.328, 154.405] to (-258.83, 323.69, -10) mm, rotated rx -180 ry 0 rz 0.01 deg; joints [38.034, -38.978, 89.114, -134.769, 60.236, 154.309]
  MoveL 609 to (-266.61, 323.69, -10) mm, rotated rx 180 ry 0 rz 0.01 deg; joints [37.868, -38.659, 88.455, -134.801, 59.921, 154.119]
  MoveC 610 to (-270.28, 324.81, -10) mm, rotated rx -180 ry 0 rz 0.01 deg; joints [37.82, -38.472, 88.069, -134.767, 59.759, 153.98] to (-272.72, 327.77, -10) mm, rotated rx 180 ry 0 rz 0.01 deg; joints [37.849, -38.277, 87.663, -134.65, 59.624, 153.791]
  MoveC 611 to (-275.16, 330.73, -10) mm, rotated rx 180 ry 0 rz 0.01 deg; joints [37.878, -38.081, 87.255, -134.531, 59.489, 153.601] to (-278.83, 331.84, -10) mm, rotated rx 180 ry 0 rz 0.01 deg; joints [37.831, -37.892, 86.864, -134.495, 59.325, 153.458]
  MoveL 612 to (-392.58, 331.84, -10) mm, rotated rx 180 ry 0 rz 0.01 deg; joints [35.559, -32.712, 76.23, -134.31, 54.385, 150.12]
  MoveC 613 to (-395.3, 330.71, -10) mm, rotated rx 180 ry 0 rz 0.01 deg; joints [35.478, -32.616, 76.034, -134.345, 54.273, 150.083] to (-396.43, 327.99, -10) mm, rotated rx 180 ry 0 rz 0.01 deg; joints [35.384, -32.654, 76.117, -134.466, 54.256, 150.18]
  MoveL 614 to (-396.42, 62.53, -10) mm, rotated rx -180 ry 0 rz 0.01 deg; joints [27.714, -40.118, 91.877, -146.46, 57.36, 161.38]
  MoveC 615 to (-395.31, 60.75, -10) mm, rotated rx 180 ry 0 rz 0.01 deg; joints [27.677, -40.207, 92.065, -146.536, 57.429, 161.468] to (-393.23, 60.98, -10) mm, rotated rx 180 ry 0 rz 0.01 deg; joints [27.719, -40.294, 92.245, -146.522, 57.521, 161.503]
  MoveC 616 to (-391.47, 62.38, -10) mm, rotated rx 180 ry 0 rz 0.01 deg; joints [27.791, -40.341, 92.338, -146.458, 57.585, 161.49] to (-389.72, 63.78, -10) mm, rotated rx -180 ry 0 rz 0.01 deg; joints [27.864, -40.386, 92.431, -146.393, 57.649, 161.476]
  MoveC 617 to (-387.84, 65.01, -10) mm, rotated rx -180 ry 0 rz 0.01 deg; joints [27.934, -40.442, 92.543, -146.335, 57.72, 161.471] to (-385.75, 65.86, -10) mm, rotated rx -180 ry 0 rz 0.01 deg; joints [27.995, -40.515, 92.692, -146.294, 57.804, 161.484]
  MoveC 618 to (-382.02, 67.04, -10) mm, rotated rx -180 ry 0 rz 0.01 deg; joints [28.095, -40.652, 92.975, -146.234, 57.959, 161.52] to (-378.32, 68.33, -10) mm, rotated rx 180 ry 0 rz 0.01 deg; joints [28.197, -40.785, 93.247, -146.169, 58.11, 161.55]
  MoveC 619 to (-374.5, 69.26, -10) mm, rotated rx 180 ry 0 rz 0.01 deg; joints [28.291, -40.93, 93.547, -146.118, 58.27, 161.595] to (-370.56, 69.33, -10) mm, rotated rx -180 ry 0 rz 0.01 deg; joints [28.36, -41.1, 93.897, -146.104, 58.443, 161.673]
  MoveC 620 to (-363.06, 68.28, -10) mm, rotated rx -180 ry 0 rz 0.01 deg; joints [28.455, -41.446, 94.618, -146.127, 58.785, 161.862] to (-355.69, 66.54, -10) mm, rotated rx 180 ry 0 rz 0.01 deg; joints [28.526, -41.8, 95.354, -146.177, 59.127, 162.069]
  MoveC 621 to (-348.73, 63.4, -10) mm, rotated rx -180 ry 0 rz 0.01 deg; joints [28.547, -42.165, 96.117, -146.286, 59.464, 162.315] to (-342.97, 58.37, -10) mm, rotated rx 180 ry 0 rz 0.01 deg; joints [28.486, -42.518, 96.859, -146.478, 59.768, 162.598]
  MoveC 622 to (-341.06, 56.18, -10) mm, rotated rx 180 ry 0 rz 0.01 deg; joints [28.449, -42.646, 97.128, -146.564, 59.874, 162.709] to (-339.11, 54.02, -10) mm, rotated rx 180 ry 0 rz 0.01 deg; joints [28.414, -42.775, 97.399, -146.648, 59.982, 162.82]
  MoveC 623 to (-337.26, 51.77, -10) mm, rotated rx 180 ry 0 rz 0.01 deg; joints [28.373, -42.9, 97.664, -146.737, 60.085, 162.931] to (-335.67, 49.32, -10) mm, rotated rx -180 ry 0 rz 0.01 deg; joints [28.322, -43.019, 97.915, -146.834, 60.18, 163.043]
  MoveL 624 to (-317.7, 18.13, -10) mm, rotated rx 180 ry 0 rz 0.01 deg; joints [27.614, -44.411, 100.869, -148.079, 61.282, 164.392]
  MoveC 625 to (-314.84, 11.63, -10) mm, rotated rx 180 ry 0 rz 0.01 deg; joints [27.447, -44.658, 101.396, -148.341, 61.472, 164.649] to (-313.46, 4.66, -10) mm, rotated rx 180 ry 0 rz 0.01 deg; joints [27.238, -44.853, 101.817, -148.633, 61.604, 164.893]
  MoveC 626 to (-313.2, -2.4, -10) mm, rotated rx 180 ry 0 rz 0.01 deg; joints [27.006, -45.003, 102.143, -148.935, 61.69, 165.12] to (-313.66, -9.46, -10) mm, rotated rx -180 ry 0 rz 0.01 deg; joints [26.76, -45.123, 102.406, -149.243, 61.744, 165.333]
  MoveC 627 to (-314.32, -12.43, -10) mm, rotated rx 180 ry 0 rz 0.01 deg; joints [26.649, -45.153, 102.475, -149.375, 61.747, 165.415] to (-315.6, -15.19, -10) mm, rotated rx 180 ry 0 rz 0.01 deg; joints [26.533, -45.155, 102.485, -149.503, 61.722, 165.48]
  MoveC 628 to (-317.08, -17.83, -10) mm, rotated rx -180 ry 0 rz 0.01 deg; joints [26.419, -45.146, 102.47, -149.627, 61.686, 165.537] to (-318.43, -20.54, -10) mm, rotated rx -180 ry 0 rz 0.01 deg; joints [26.304, -45.143, 102.47, -149.752, 61.657, 165.599]
  MoveC 629 to (-318.28, -22.81, -10) mm, rotated rx -180 ry 0 rz 0.01 deg; joints [26.23, -45.192, 102.577, -149.85, 61.687, 165.672] to (-316.28, -23.91, -10) mm, rotated rx 180 ry 0 rz 0.01 deg; joints [26.226, -45.294, 102.791, -149.884, 61.783, 165.738]
  MoveL 630 to (-77.2, -23.91, -10) mm, rotated rx -180 ry 0 rz 0.01 deg; joints [30.885, -54.011, 121.229, -147.149, 71.2, 169.254]
  MoveC 631 to (-75.22, -22.81, -10) mm, rotated rx 180 ry 0 rz 0.01 deg; joints [30.972, -54.056, 121.323, -147.069, 71.259, 169.252] to (-75.11, -20.54, -10) mm, rotated rx -180 ry 0 rz 0.01 deg; joints [31.06, -54.017, 121.234, -146.969, 71.236, 169.194]
  MoveC 632 to (-76.72, -17.22, -10) mm, rotated rx 180 ry 0 rz 0.01 deg; joints [31.148, -53.902, 120.979, -146.851, 71.137, 169.083] to (-78.3, -13.88, -10) mm, rotated rx -180 ry 0 rz 0.01 deg; joints [31.238, -53.786, 120.724, -146.733, 71.04, 168.971]
  MoveC 633 to (-79.57, -10.4, -10) mm, rotated rx 180 ry 0 rz 0.01 deg; joints [31.339, -53.678, 120.484, -146.603, 70.951, 168.859] to (-80.25, -6.75, -10) mm, rotated rx 180 ry 0 rz 0.01 deg; joints [31.459, -53.586, 120.279, -146.457, 70.883, 168.751]
  MoveC 634 to (-80.53, -3.18, -10) mm, rotated rx 180 ry 0 rz 0.01 deg; joints [31.586, -53.508, 120.104, -146.308, 70.83, 168.65] to (-80.67, 0.4, -10) mm, rotated rx 180 ry 0 rz 0.01 deg; joints [31.715, -53.435, 119.938, -146.156, 70.782, 168.55]
  MoveC 635 to (-80.48, 3.98, -10) mm, rotated rx 180 ry 0 rz 0.01 deg; joints [31.852, -53.372, 119.795, -145.999, 70.746, 168.455] to (-79.78, 7.5, -10) mm, rotated rx 180 ry 0 rz 0.01 deg; joints [31.998, -53.326, 119.69, -145.837, 70.729, 168.368]
  MoveC 636 to (-78.05, 12.87, -10) mm, rotated rx -180 ry 0 rz 0.01 deg; joints [32.235, -53.278, 119.575, -145.579, 70.728, 168.245] to (-75.85, 18.05, -10) mm, rotated rx -180 ry 0 rz 0.01 deg; joints [32.476, -53.247, 119.498, -145.322, 70.745, 168.133]
  MoveL 637 to (-57.49, 49.9, -10) mm, rotated rx 180 ry 0 rz 0.01 deg; joints [34.066, -53.197, 119.323, -143.661, 71.016, 167.503]
  MoveC 638 to (-53.21, 55.79, -10) mm, rotated rx 180 ry 0 rz 0.01 deg; joints [34.381, -53.212, 119.342, -143.339, 71.095, 167.397] to (-47.8, 60.66, -10) mm, rotated rx 180 ry 0 rz 0.01 deg; joints [34.688, -53.283, 119.483, -143.039, 71.226, 167.337]
  MoveC 639 to (-41.68, 64.55, -10) mm, rotated rx 180 ry 0 rz 0.01 deg; joints [34.978, -53.396, 119.718, -142.766, 71.393, 167.316] to (-35.11, 67.63, -10) mm, rotated rx -180 ry 0 rz 0.01 deg; joints [35.252, -53.539, 120.017, -142.518, 71.583, 167.324]
  MoveC 640 to (-31.36, 68.77, -10) mm, rotated rx 180 ry 0 rz 0.01 deg; joints [35.387, -53.633, 120.217, -142.401, 71.7, 167.347] to (-27.47, 69.27, -10) mm, rotated rx 180 ry 0 rz 0.01 deg; joints [35.503, -53.745, 120.455, -142.307, 71.829, 167.39]
  MoveC 641 to (-23.56, 69.37, -10) mm, rotated rx 180 ry 0 rz 0.01 deg; joints [35.607, -53.866, 120.714, -142.23, 71.962, 167.445] to (-19.64, 69.3, -10) mm, rotated rx 180 ry 0 rz 0.01 deg; joints [35.704, -53.99, 120.98, -142.158, 72.098, 167.504]
  MoveC 642 to (-15.49, 68.8, -10) mm, rotated rx -180 ry 0 rz 0.01 deg; joints [35.793, -54.131, 121.283, -142.1, 72.247, 167.58] to (-11.46, 67.64, -10) mm, rotated rx -180 ry 0 rz 0.01 deg; joints [35.856, -54.281, 121.608, -142.07, 72.4, 167.673]
  MoveC 643 to (-7.62, 65.98, -10) mm, rotated rx -180 ry 0 rz 0.01 deg; joints [35.896, -54.436, 121.944, -142.065, 72.552, 167.777] to (-3.95, 63.99, -10) mm, rotated rx 180 ry 0 rz 0.01 deg; joints [35.92, -54.592, 122.284, -142.075, 72.703, 167.888]
  MoveC 644 to (-2.96, 63.32, -10) mm, rotated rx -180 ry 0 rz 0.01 deg; joints [35.921, -54.637, 122.382, -142.084, 72.745, 167.921] to (-2.06, 62.55, -10) mm, rotated rx 180 ry 0 rz 0.01 deg; joints [35.917, -54.681, 122.479, -142.098, 72.786, 167.957]
  MoveC 645 to (-1.18, 61.74, -10) mm, rotated rx 180 ry 0 rz 0.01 deg; joints [35.911, -54.725, 122.576, -142.115, 72.826, 167.992] to (-0.27, 60.98, -10) mm, rotated rx 180 ry 0 rz 0.01 deg; joints [35.907, -54.77, 122.673, -142.128, 72.867, 168.027]
  MoveC 646 to (1.8, 60.74, -10) mm, rotated rx -180 ry 0 rz 0.01 deg; joints [35.953, -54.839, 122.821, -142.097, 72.94, 168.065] to (2.91, 62.51, -10) mm, rotated rx 180 ry 0 rz 0.01 deg; joints [36.046, -54.835, 122.81, -142.001, 72.956, 168.031]
  MoveL 647 to (2.91, 328, -10) mm, rotated rx -180 ry 0 rz 0.01 deg; joints [44.538, -48.111, 108.073, -131.574, 69.676, 159.387]
  MoveC 648 to (1.78, 330.72, -10) mm, rotated rx 180 ry 0 rz 0.01 deg; joints [44.583, -47.996, 107.828, -131.493, 69.607, 159.267] to (-0.95, 331.85, -10) mm, rotated rx -180 ry 0 rz 0.01 deg; joints [44.539, -47.879, 107.581, -131.5, 69.504, 159.179]
  MoveL 649 to (-150.16, 331.85, -10) mm, rotated rx 180 ry 0 rz 0.01 deg; joints [40.714, -42.901, 97.21, -133.619, 64.323, 156.395]
  MoveC 650 to (-151.8, 330.74, -10) mm, rotated rx 180 ry 0 rz 0.01 deg; joints [40.645, -42.875, 97.158, -133.681, 64.275, 156.405] to (-151.39, 328.8, -10) mm, rotated rx 180 ry 0 rz 0.01 deg; joints [40.6, -42.949, 97.313, -133.753, 64.313, 156.491]
  MoveC 651 to (-145.42, 321.36, -10) mm, rotated rx 180 ry 0 rz 0.01 deg; joints [40.536, -43.388, 98.235, -133.985, 64.62, 156.905] to (-141.44, 312.68, -10) mm, rotated rx 180 ry 0 rz 0.01 deg; joints [40.388, -43.788, 99.078, -134.284, 64.868, 157.322]
  MoveC 652 to (-140.19, 308.37, -10) mm, rotated rx 180 ry 0 rz 0.01 deg; joints [40.296, -43.96, 99.441, -134.441, 64.964, 157.513] to (-139.22, 303.98, -10) mm, rotated rx -180 ry 0 rz 0.01 deg; joints [40.195, -44.123, 99.786, -134.603, 65.052, 157.701]
  MoveC 653 to (-138.85, 299.48, -10) mm, rotated rx -180 ry 0 rz 0.01 deg; joints [40.076, -44.267, 100.093, -134.777, 65.118, 157.88] to (-139.43, 295.01, -10) mm, rotated rx 180 ry 0 rz 0.01 deg; joints [39.934, -44.376, 100.327, -134.961, 65.15, 158.039]
  MoveC 654 to (-141.37, 287.94, -10) mm, rotated rx -180 ry 0 rz 0.01 deg; joints [39.685, -44.511, 100.618, -135.264, 65.162, 158.269] to (-143.78, 281.01, -10) mm, rotated rx -180 ry 0 rz 0.01 deg; joints [39.428, -44.623, 100.862, -135.568, 65.156, 158.483]
  MoveC 655 to (-147.4, 274.56, -10) mm, rotated rx 180 ry 0 rz 0.01 deg; joints [39.156, -44.678, 100.985, -135.867, 65.099, 158.656] to (-152.66, 269.36, -10) mm, rotated rx 180 ry 0 rz 0.01 deg; joints [38.88, -44.636, 100.906, -136.135, 64.966, 158.749]
  MoveC 656 to (-158.72, 265.42, -10) mm, rotated rx -180 ry 0 rz 0.01 deg; joints [38.624, -44.529, 100.69, -136.361, 64.789, 158.779] to (-165.21, 262.26, -10) mm, rotated rx -180 ry 0 rz 0.01 deg; joints [38.381, -44.383, 100.392, -136.56, 64.585, 158.771]
  MoveC 657 to (-172.14, 260.16, -10) mm, rotated rx 180 ry 0 rz 0.01 deg; joints [38.159, -44.19, 99.993, -136.719, 64.35, 158.715] to (-179.34, 259.46, -10) mm, rotated rx 180 ry 0 rz 0.01 deg; joints [37.974, -43.946, 99.488, -136.823, 64.088, 158.601]
  MoveL 658 to (-214.9, 259.46, -10) mm, rotated rx -180 ry 0 rz 0.01 deg; joints [37.177, -42.616, 96.727, -137.153, 62.729, 157.885]
  MoveC 659 to (-222.2, 260.21, -10) mm, rotated rx 180 ry 0 rz 0.01 deg; joints [37.039, -42.315, 96.103, -137.182, 62.436, 157.704] to (-229.19, 262.43, -10) mm, rotated rx 180 ry 0 rz 0.01 deg; joints [36.951, -41.983, 95.41, -137.144, 62.137, 157.471]
  MoveC 660 to (-235.69, 265.79, -10) mm, rotated rx 180 ry 0 rz 0.01 deg; joints [36.907, -41.634, 94.683, -137.053, 61.842, 157.201] to (-241.65, 270.03, -10) mm, rotated rx 180 ry 0 rz 0.01 deg; joints [36.9, -41.278, 93.941, -136.918, 61.556, 156.905]
  MoveC 661 to (-245.62, 274.01, -10) mm, rotated rx 180 ry 0 rz 0.01 deg; joints [36.929, -41.006, 93.372, -136.778, 61.352, 156.66] to (-248.74, 278.69, -10) mm, rotated rx -180 ry 0 rz 0.01 deg; joints [36.995, -40.746, 92.828, -136.602, 61.173, 156.404]
  MoveC 662 to (-251.05, 283.79, -10) mm, rotated rx 180 ry 0 rz 0.01 deg; joints [37.09, -40.504, 92.32, -136.403, 61.021, 156.146] to (-252.71, 289.15, -10) mm, rotated rx 180 ry 0 rz 0.01 deg; joints [37.206, -40.279, 91.848, -136.189, 60.891, 155.891]
  MoveC 663 to (-253.97, 299.77, -10) mm, rotated rx 180 ry 0 rz 0.01 deg; joints [37.476, -39.91, 91.071, -135.751, 60.715, 155.427] to (-252.7, 310.39, -10) mm, rotated rx 180 ry 0 rz 0.01 deg; joints [37.799, -39.639, 90.496, -135.299, 60.64, 155.017]
  MoveC 664 to (-248.72, 320.35, -10) mm, rotated rx -180 ry 0 rz 0.01 deg; joints [38.159, -39.493, 90.18, -134.862, 60.681, 154.694] to (-242.11, 328.8, -10) mm, rotated rx 180 ry 0 rz 0.01 deg; joints [38.535, -39.496, 90.174, -134.474, 60.844, 154.495]
  MoveC 665 to (-241.7, 330.74, -10) mm, rotated rx 180 ry 0 rz 0.01 deg; joints [38.597, -39.452, 90.08, -134.391, 60.838, 154.423] to (-243.34, 331.84, -10) mm, rotated rx -180 ry 0 rz 0.01 deg; joints [38.591, -39.351, 89.871, -134.353, 60.759, 154.337]
  MoveL 666 to (-278.83, 331.84, -10) mm, rotated rx -180 ry 0 rz 0.01 deg; joints [37.831, -37.892, 86.864, -134.495, 59.325, 153.458]
  MoveL 667 to (-279.44, 331.69, -9.83) mm, rotated rx 180 ry 0 rz 0.01 deg; joints [37.814, -37.879, 86.822, -134.5, 59.297, 153.444]
  MoveL 668 to (-279.8, 331.4, -9.37) mm, rotated rx 180 ry 0 rz 0.01 deg; joints [37.798, -37.894, 86.812, -134.506, 59.272, 153.431]
  MoveL 669 to (-279.9, 331.26, -8.73) mm, rotated rx 180 ry 0 rz 0.01 deg; joints [37.792, -37.922, 86.814, -134.501, 59.25, 153.412]
  Set speed (500.0 mm/s)
  MoveL 670 to (-279.9, 331.26, 11.77) mm, rotated rx -180 ry 0 rz 0.01 deg; joints [37.783, -38.83, 86.849, -134.134, 58.636, 152.688]
  Set speed (500.0 mm/s)
  MoveL 671 to (-398.5, 339.2, 11.77) mm, rotated rx -180 ry 0 rz 0.01 deg; joints [35.632, -33.057, 75.127, -133.473, 53.419, 148.782]
  Set speed (100.0 mm/s)
  MoveL 672 to (-398.51, 339.2, 11.68) mm, rotated rx 180 ry 0 rz 0.01 deg; joints [35.632, -33.053, 75.127, -133.475, 53.422, 148.786]
  MoveL 673 to (-398.63, 339.2, 11.21) mm, rotated rx -180 ry 0 rz 0.01 deg; joints [35.63, -33.028, 75.114, -133.484, 53.429, 148.798]
  MoveL 674 to (-398.92, 339.18, 10.83) mm, rotated rx -180 ry 0 rz 0.01 deg; joints [35.624, -32.998, 75.084, -133.49, 53.426, 148.802]
  MoveL 675 to (-399.34, 339.13, 10.58) mm, rotated rx 180 ry 0 rz 0.01 deg; joints [35.615, -32.969, 75.045, -133.494, 53.415, 148.799]
  MoveL 676 to (-399.69, 339.08, 10.5) mm, rotated rx -180 ry 0 rz 0.01 deg; joints [35.607, -32.949, 75.013, -133.496, 53.401, 148.792]
  MoveL 677 to (-399.72, 339.07, 10.5) mm, rotated rx -180 ry 0 rz 0.01 deg; joints [35.606, -32.948, 75.01, -133.496, 53.4, 148.791]
  MoveL 678 to (-400.55, 338.85, 10.47) mm, rotated rx -180 ry 0 rz 0.01 deg; joints [35.584, -32.913, 74.941, -133.5, 53.365, 148.775]
  MoveL 679 to (-400.6, 338.83, 10.47) mm, rotated rx -180 ry 0 rz 0.01 deg; joints [35.583, -32.911, 74.938, -133.5, 53.363, 148.774]
  MoveL 680 to (-401.28, 338.49, 10.44) mm, rotated rx -180 ry 0 rz 0.01 deg; joints [35.561, -32.887, 74.892, -133.511, 53.337, 148.768]
  MoveL 681 to (-401.4, 338.42, 10.44) mm, rotated rx 180 ry 0 rz 0.01 deg; joints [35.557, -32.883, 74.885, -133.514, 53.332, 148.768]
  MoveL 682 to (-402.84, 337.05, 10.37) mm, rotated rx 180 ry 0 rz 0.01 deg; joints [35.494, -32.856, 74.837, -133.569, 53.284, 148.789]
  MoveL 683 to (-402.87, 337.02, 10.37) mm, rotated rx -180 ry 0 rz 0.01 deg; joints [35.493, -32.856, 74.837, -133.571, 53.283, 148.79]
  MoveL 684 to (-403.75, 334.43, 10.27) mm, rotated rx -180 ry 0 rz 0.01 deg; joints [35.408, -32.899, 74.935, -133.69, 53.276, 148.895]
  MoveL 685 to (-403.78, 333.95, 10.25) mm, rotated rx 180 ry 0 rz 0.01 deg; joints [35.395, -32.914, 74.968, -133.713, 53.281, 148.919]
  MoveL 686 to (-403.79, 333.65, 10.24) mm, rotated rx 180 ry 0 rz 0.01 deg; joints [35.387, -32.924, 74.989, -133.728, 53.284, 148.934]
  MoveL 687 to (-403.79, 333.05, 10.22) mm, rotated rx -180 ry 0 rz 0.01 deg; joints [35.371, -32.944, 75.033, -133.757, 53.292, 148.966]
  MoveL 688 to (-401.25, 328.08, 10.02) mm, rotated rx 180 ry 0 rz 0.01 deg; joints [35.287, -33.24, 75.657, -134.021, 53.475, 149.314]
  MoveL 689 to (-395.74, 327.2, 9.82) mm, rotated rx -180 ry 0 rz 0.01 deg; joints [35.368, -33.54, 76.283, -134.109, 53.744, 149.554]
  MoveL 690 to (-391.79, 331.15, 9.61) mm, rotated rx -180 ry 0 rz 0.01 deg; joints [35.547, -33.591, 76.398, -133.954, 53.883, 149.497]
  MoveL 691 to (-392.66, 336.66, 9.41) mm, rotated rx -180 ry 0 rz 0.01 deg; joints [35.676, -33.345, 75.908, -133.689, 53.783, 149.198]
  MoveL 692 to (-397.64, 339.2, 9.21) mm, rotated rx -180 ry 0 rz 0.01 deg; joints [35.649, -32.996, 75.214, -133.534, 53.53, 148.904]
  MoveL 693 to (-398.51, 339.2, 9.18) mm, rotated rx -180 ry 0 rz 0.01 deg; joints [35.633, -32.951, 75.124, -133.527, 53.491, 148.875]
  MoveL 694 to (-399.34, 339.13, 9.15) mm, rotated rx -180 ry 0 rz 0.01 deg; joints [35.615, -32.91, 75.044, -133.524, 53.454, 148.85]
  MoveL 695 to (-399.69, 339.08, 9.14) mm, rotated rx -180 ry 0 rz 0.01 deg; joints [35.607, -32.894, 75.011, -133.524, 53.439, 148.841]
  MoveL 696 to (-400.55, 338.85, 9.11) mm, rotated rx -180 ry 0 rz 0.01 deg; joints [35.585, -32.857, 74.939, -133.529, 53.403, 148.823]
  MoveL 697 to (-400.6, 338.83, 9.1) mm, rotated rx -180 ry 0 rz 0.01 deg; joints [35.584, -32.855, 74.936, -133.529, 53.401, 148.823]
  MoveL 698 to (-401.28, 338.49, 9.08) mm, rotated rx 180 ry 0 rz 0.01 deg; joints [35.562, -32.831, 74.89, -133.54, 53.374, 148.817]
  MoveL 699 to (-401.4, 338.42, 9.07) mm, rotated rx 180 ry 0 rz 0.01 deg; joints [35.558, -32.827, 74.883, -133.543, 53.37, 148.817]
  MoveL 700 to (-402.84, 337.05, 9) mm, rotated rx 180 ry 0 rz 0.01 deg; joints [35.495, -32.8, 74.835, -133.598, 53.322, 148.838]
  MoveL 701 to (-402.87, 337.02, 9) mm, rotated rx -180 ry 0 rz 0.01 deg; joints [35.493, -32.8, 74.835, -133.599, 53.321, 148.839]
  MoveL 702 to (-403.75, 334.43, 8.9) mm, rotated rx 180 ry 0 rz 0.01 deg; joints [35.409, -32.843, 74.934, -133.719, 53.314, 148.943]
  MoveL 703 to (-403.78, 333.95, 8.89) mm, rotated rx -180 ry 0 rz 0.01 deg; joints [35.395, -32.858, 74.967, -133.742, 53.319, 148.968]
  MoveL 704 to (-403.79, 333.65, 8.88) mm, rotated rx -180 ry 0 rz 0.01 deg; joints [35.387, -32.868, 74.987, -133.756, 53.322, 148.983]
  MoveL 705 to (-403.79, 333.05, 8.86) mm, rotated rx -180 ry 0 rz 0.01 deg; joints [35.371, -32.888, 75.032, -133.786, 53.33, 149.014]
  MoveL 706 to (-401.25, 328.08, 8.65) mm, rotated rx -180 ry 0 rz 0.01 deg; joints [35.288, -33.184, 75.655, -134.05, 53.513, 149.362]
  MoveL 707 to (-395.74, 327.2, 8.45) mm, rotated rx 180 ry 0 rz 0.01 deg; joints [35.368, -33.484, 76.281, -134.137, 53.783, 149.602]
  MoveL 708 to (-391.79, 331.15, 8.25) mm, rotated rx -180 ry 0 rz 0.01 deg; joints [35.548, -33.535, 76.396, -133.982, 53.922, 149.546]
  MoveL 709 to (-392.66, 336.66, 8.05) mm, rotated rx -180 ry 0 rz 0.01 deg; joints [35.677, -33.289, 75.907, -133.718, 53.821, 149.246]
  MoveL 710 to (-397.64, 339.2, 7.84) mm, rotated rx -180 ry 0 rz 0.01 deg; joints [35.65, -32.94, 75.212, -133.562, 53.568, 148.953]
  MoveL 711 to (-398.51, 339.2, 7.81) mm, rotated rx -180 ry 0 rz 0.01 deg; joints [35.633, -32.895, 75.123, -133.556, 53.529, 148.923]
  MoveL 712 to (-399.34, 339.13, 7.78) mm, rotated rx 180 ry 0 rz 0.01 deg; joints [35.616, -32.854, 75.042, -133.553, 53.492, 148.899]
  MoveL 713 to (-399.69, 339.08, 7.77) mm, rotated rx -180 ry 0 rz 0.01 deg; joints [35.608, -32.838, 75.009, -133.553, 53.477, 148.889]
  MoveL 714 to (-400.55, 338.85, 7.74) mm, rotated rx -180 ry 0 rz 0.01 deg; joints [35.586, -32.801, 74.938, -133.557, 53.44, 148.872]
  MoveL 715 to (-400.6, 338.83, 7.74) mm, rotated rx -180 ry 0 rz 0.01 deg; joints [35.584, -32.799, 74.934, -133.558, 53.439, 148.871]
  MoveL 716 to (-401.28, 338.49, 7.71) mm, rotated rx -180 ry 0 rz 0.01 deg; joints [35.563, -32.775, 74.888, -133.569, 53.412, 148.865]
  MoveL 717 to (-401.4, 338.42, 7.71) mm, rotated rx 180 ry 0 rz 0.01 deg; joints [35.558, -32.772, 74.881, -133.571, 53.407, 148.865]
  MoveL 718 to (-402.84, 337.05, 7.64) mm, rotated rx -180 ry 0 rz 0.01 deg; joints [35.495, -32.744, 74.833, -133.626, 53.359, 148.887]
  MoveL 719 to (-402.87, 337.02, 7.64) mm, rotated rx -180 ry 0 rz 0.01 deg; joints [35.494, -32.744, 74.833, -133.628, 53.359, 148.888]
  MoveL 720 to (-403.75, 334.43, 7.54) mm, rotated rx -180 ry 0 rz 0.01 deg; joints [35.409, -32.787, 74.932, -133.747, 53.351, 148.992]
  MoveL 721 to (-403.78, 333.95, 7.52) mm, rotated rx 180 ry 0 rz 0.01 deg; joints [35.396, -32.802, 74.965, -133.771, 53.357, 149.016]
  MoveL 722 to (-403.79, 333.65, 7.51) mm, rotated rx -180 ry 0 rz 0.01 deg; joints [35.388, -32.812, 74.986, -133.785, 53.36, 149.031]
  MoveL 723 to (-403.79, 333.05, 7.49) mm, rotated rx -180 ry 0 rz 0.01 deg; joints [35.372, -32.832, 75.03, -133.814, 53.368, 149.063]
  MoveL 724 to (-401.25, 328.08, 7.29) mm, rotated rx -180 ry 0 rz 0.01 deg; joints [35.288, -33.128, 75.654, -134.078, 53.551, 149.41]
  MoveL 725 to (-395.74, 327.2, 7.09) mm, rotated rx -180 ry 0 rz 0.01 deg; joints [35.369, -33.428, 76.28, -134.165, 53.821, 149.65]
  MoveL 726 to (-391.79, 331.15, 6.88) mm, rotated rx -180 ry 0 rz 0.01 deg; joints [35.548, -33.479, 76.395, -134.01, 53.96, 149.594]
  MoveL 727 to (-392.66, 336.66, 6.68) mm, rotated rx -180 ry 0 rz 0.01 deg; joints [35.678, -33.233, 75.905, -133.746, 53.859, 149.295]
  MoveL 728 to (-397.64, 339.2, 6.48) mm, rotated rx 180 ry 0 rz 0.01 deg; joints [35.65, -32.884, 75.21, -133.59, 53.606, 149.001]
  MoveL 729 to (-398.51, 339.2, 6.45) mm, rotated rx -180 ry 0 rz 0.01 deg; joints [35.634, -32.839, 75.121, -133.584, 53.566, 148.972]
  MoveL 730 to (-399.34, 339.13, 6.42) mm, rotated rx 180 ry 0 rz 0.01 deg; joints [35.617, -32.798, 75.04, -133.581, 53.53, 148.947]
  MoveL 731 to (-399.69, 339.08, 6.41) mm, rotated rx -180 ry 0 rz 0.01 deg; joints [35.608, -32.782, 75.008, -133.581, 53.514, 148.938]
  MoveL 732 to (-400.55, 338.85, 6.38) mm, rotated rx -180 ry 0 rz 0.01 deg; joints [35.586, -32.745, 74.936, -133.586, 53.478, 148.92]
  MoveL 733 to (-400.6, 338.83, 6.37) mm, rotated rx -180 ry 0 rz 0.01 deg; joints [35.585, -32.743, 74.932, -133.586, 53.476, 148.92]
  MoveL 734 to (-401.28, 338.49, 6.35) mm, rotated rx -180 ry 0 rz 0.01 deg; joints [35.563, -32.719, 74.887, -133.597, 53.45, 148.914]
  MoveL 735 to (-401.4, 338.42, 6.34) mm, rotated rx -180 ry 0 rz 0.01 deg; joints [35.559, -32.716, 74.879, -133.6, 53.445, 148.913]
  MoveL 736 to (-402.84, 337.05, 6.27) mm, rotated rx 180 ry 0 rz 0.01 deg; joints [35.496, -32.688, 74.831, -133.655, 53.397, 148.935]
  MoveL 737 to (-402.87, 337.02, 6.27) mm, rotated rx -180 ry 0 rz 0.01 deg; joints [35.495, -32.688, 74.831, -133.656, 53.396, 148.936]
  MoveL 738 to (-403.75, 334.43, 6.17) mm, rotated rx -180 ry 0 rz 0.01 deg; joints [35.41, -32.731, 74.93, -133.776, 53.389, 149.04]
  MoveL 739 to (-403.78, 333.95, 6.16) mm, rotated rx -180 ry 0 rz 0.01 deg; joints [35.396, -32.746, 74.963, -133.799, 53.394, 149.065]
  MoveL 740 to (-403.79, 333.65, 6.15) mm, rotated rx -180 ry 0 rz 0.01 deg; joints [35.389, -32.756, 74.984, -133.813, 53.398, 149.08]
  MoveL 741 to (-403.79, 333.05, 6.13) mm, rotated rx -180 ry 0 rz 0.01 deg; joints [35.373, -32.776, 75.028, -133.843, 53.406, 149.111]
  MoveL 742 to (-401.25, 328.08, 5.92) mm, rotated rx -180 ry 0 rz 0.01 deg; joints [35.289, -33.072, 75.652, -134.106, 53.589, 149.459]
  MoveL 743 to (-395.74, 327.2, 5.72) mm, rotated rx -180 ry 0 rz 0.01 deg; joints [35.369, -33.371, 76.278, -134.193, 53.859, 149.698]
  MoveL 744 to (-391.79, 331.15, 5.52) mm, rotated rx -180 ry 0 rz 0.01 deg; joints [35.549, -33.422, 76.393, -134.038, 53.998, 149.642]
  MoveL 745 to (-392.66, 336.66, 5.32) mm, rotated rx 180 ry 0 rz 0.01 deg; joints [35.678, -33.177, 75.903, -133.774, 53.897, 149.343]
  MoveL 746 to (-397.64, 339.2, 5.11) mm, rotated rx -180 ry 0 rz 0.01 deg; joints [35.651, -32.828, 75.208, -133.619, 53.643, 149.049]
  MoveL 747 to (-398.51, 339.2, 5.08) mm, rotated rx -180 ry 0 rz 0.01 deg; joints [35.635, -32.783, 75.119, -133.612, 53.604, 149.02]
  MoveL 748 to (-399.34, 339.13, 5.06) mm, rotated rx -180 ry 0 rz 0.01 deg; joints [35.617, -32.742, 75.038, -133.609, 53.567, 148.995]
  MoveL 749 to (-399.69, 339.08, 5.04) mm, rotated rx -180 ry 0 rz 0.01 deg; joints [35.609, -32.726, 75.006, -133.609, 53.552, 148.986]
  MoveL 750 to (-400.55, 338.85, 5.01) mm, rotated rx 180 ry 0 rz 0.01 deg; joints [35.587, -32.689, 74.934, -133.614, 53.516, 148.969]
  MoveL 751 to (-400.6, 338.83, 5.01) mm, rotated rx -180 ry 0 rz 0.01 deg; joints [35.586, -32.687, 74.93, -133.614, 53.514, 148.968]
  MoveL 752 to (-401.28, 338.49, 4.98) mm, rotated rx -180 ry 0 rz 0.01 deg; joints [35.564, -32.663, 74.885, -133.625, 53.487, 148.962]
  MoveL 753 to (-401.4, 338.42, 4.98) mm, rotated rx -180 ry 0 rz 0.01 deg; joints [35.559, -32.66, 74.877, -133.628, 53.482, 148.962]
  MoveL 754 to (-402.84, 337.05, 4.91) mm, rotated rx -180 ry 0 rz 0.01 deg; joints [35.497, -32.632, 74.829, -133.683, 53.434, 148.983]
  MoveL 755 to (-402.87, 337.02, 4.91) mm, rotated rx 180 ry 0 rz 0.01 deg; joints [35.495, -32.632, 74.829, -133.685, 53.434, 148.984]
  MoveL 756 to (-403.75, 334.43, 4.81) mm, rotated rx -180 ry 0 rz 0.01 deg; joints [35.41, -32.675, 74.928, -133.804, 53.427, 149.088]
  MoveL 757 to (-403.78, 333.95, 4.79) mm, rotated rx -180 ry 0 rz 0.01 deg; joints [35.397, -32.69, 74.961, -133.827, 53.432, 149.113]
  MoveL 758 to (-403.79, 333.65, 4.78) mm, rotated rx 180 ry 0 rz 0.01 deg; joints [35.389, -32.7, 74.982, -133.842, 53.436, 149.128]
  MoveL 759 to (-403.79, 333.05, 4.76) mm, rotated rx 180 ry 0 rz 0.01 deg; joints [35.373, -32.72, 75.026, -133.871, 53.444, 149.159]
  MoveL 760 to (-401.25, 328.08, 4.56) mm, rotated rx 180 ry 0 rz 0.01 deg; joints [35.289, -33.016, 75.65, -134.134, 53.627, 149.506]
  MoveL 761 to (-395.74, 327.2, 4.36) mm, rotated rx -180 ry 0 rz 0.01 deg; joints [35.37, -33.315, 76.276, -134.221, 53.897, 149.746]
  MoveL 762 to (-391.79, 331.15, 4.15) mm, rotated rx 180 ry 0 rz 0.01 deg; joints [35.549, -33.366, 76.391, -134.066, 54.036, 149.69]
  MoveL 763 to (-392.66, 336.66, 3.95) mm, rotated rx 180 ry 0 rz 0.01 deg; joints [35.679, -33.12, 75.901, -133.802, 53.935, 149.391]
  MoveL 764 to (-397.64, 339.2, 3.75) mm, rotated rx 180 ry 0 rz 0.01 deg; joints [35.652, -32.772, 75.206, -133.647, 53.681, 149.098]
  MoveL 765 to (-398.51, 339.2, 3.72) mm, rotated rx 180 ry 0 rz 0.01 deg; joints [35.635, -32.727, 75.117, -133.641, 53.642, 149.068]
  MoveL 766 to (-399.34, 339.13, 3.69) mm, rotated rx -180 ry 0 rz 0.01 deg; joints [35.618, -32.686, 75.036, -133.638, 53.605, 149.044]
  MoveL 767 to (-399.69, 339.08, 3.68) mm, rotated rx -180 ry 0 rz 0.01 deg; joints [35.61, -32.67, 75.003, -133.638, 53.589, 149.034]
  MoveL 768 to (-400.55, 338.85, 3.65) mm, rotated rx -180 ry 0 rz 0.01 deg; joints [35.587, -32.633, 74.931, -133.642, 53.553, 149.017]
  MoveL 769 to (-400.6, 338.83, 3.65) mm, rotated rx -180 ry 0 rz 0.01 deg; joints [35.586, -32.631, 74.928, -133.643, 53.551, 149.016]
  MoveL 770 to (-401.28, 338.49, 3.62) mm, rotated rx -180 ry 0 rz 0.01 deg; joints [35.564, -32.607, 74.882, -133.654, 53.525, 149.01]
  MoveL 771 to (-401.4, 338.42, 3.61) mm, rotated rx 180 ry 0 rz 0.01 deg; joints [35.56, -32.603, 74.875, -133.656, 53.52, 149.01]
  MoveL 772 to (-402.84, 337.05, 3.54) mm, rotated rx -180 ry 0 rz 0.01 deg; joints [35.497, -32.576, 74.827, -133.712, 53.472, 149.031]
  MoveL 773 to (-402.87, 337.02, 3.54) mm, rotated rx -180 ry 0 rz 0.01 deg; joints [35.496, -32.576, 74.827, -133.713, 53.471, 149.032]
  MoveL 774 to (-403.75, 334.43, 3.45) mm, rotated rx -180 ry 0 rz 0.01 deg; joints [35.411, -32.619, 74.926, -133.832, 53.465, 149.136]
  MoveL 775 to (-403.78, 333.95, 3.43) mm, rotated rx -180 ry 0 rz 0.01 deg; joints [35.398, -32.634, 74.959, -133.856, 53.47, 149.161]
  MoveL 776 to (-403.79, 333.65, 3.42) mm, rotated rx -180 ry 0 rz 0.01 deg; joints [35.39, -32.644, 74.979, -133.87, 53.473, 149.176]
  MoveL 777 to (-403.79, 333.05, 3.4) mm, rotated rx -180 ry 0 rz 0.01 deg; joints [35.374, -32.664, 75.024, -133.899, 53.481, 149.207]
  MoveL 778 to (-401.25, 328.08, 3.2) mm, rotated rx -180 ry 0 rz 0.01 deg; joints [35.29, -32.959, 75.647, -134.162, 53.665, 149.554]
  MoveL 779 to (-395.74, 327.2, 2.99) mm, rotated rx -180 ry 0 rz 0.01 deg; joints [35.371, -33.258, 76.273, -134.249, 53.936, 149.794]
  MoveL 780 to (-391.79, 331.15, 2.79) mm, rotated rx -180 ry 0 rz 0.01 deg; joints [35.55, -33.309, 76.388, -134.093, 54.074, 149.738]
  MoveL 781 to (-392.66, 336.66, 2.59) mm, rotated rx 180 ry 0 rz 0.01 deg; joints [35.679, -33.064, 75.899, -133.829, 53.973, 149.439]
  MoveL 782 to (-397.64, 339.2, 2.39) mm, rotated rx -180 ry 0 rz 0.01 deg; joints [35.652, -32.716, 75.204, -133.675, 53.718, 149.146]
  MoveL 783 to (-398.51, 339.2, 2.36) mm, rotated rx -180 ry 0 rz 0.01 deg; joints [35.636, -32.671, 75.114, -133.669, 53.679, 149.116]
  MoveL 784 to (-399.34, 339.13, 2.33) mm, rotated rx 180 ry 0 rz 0.01 deg; joints [35.618, -32.63, 75.034, -133.666, 53.642, 149.092]
  MoveL 785 to (-399.69, 339.08, 2.31) mm, rotated rx -180 ry 0 rz 0.01 deg; joints [35.61, -32.613, 75.001, -133.666, 53.627, 149.082]
  MoveL 786 to (-400.55, 338.85, 2.28) mm, rotated rx -180 ry 0 rz 0.01 deg; joints [35.588, -32.577, 74.929, -133.67, 53.591, 149.065]
  MoveL 787 to (-400.6, 338.83, 2.28) mm, rotated rx 180 ry 0 rz 0.01 deg; joints [35.587, -32.575, 74.926, -133.671, 53.589, 149.064]
  MoveL 788 to (-401.28, 338.49, 2.25) mm, rotated rx 180 ry 0 rz 0.01 deg; joints [35.565, -32.551, 74.88, -133.682, 53.562, 149.058]
  MoveL 789 to (-401.4, 338.42, 2.25) mm, rotated rx -180 ry 0 rz 0.01 deg; joints [35.561, -32.547, 74.873, -133.685, 53.557, 149.058]
  MoveL 790 to (-402.84, 337.05, 2.18) mm, rotated rx -180 ry 0 rz 0.01 deg; joints [35.498, -32.52, 74.825, -133.74, 53.509, 149.079]
  MoveL 791 to (-402.87, 337.02, 2.18) mm, rotated rx -180 ry 0 rz 0.01 deg; joints [35.496, -32.52, 74.825, -133.741, 53.509, 149.08]
  MoveL 792 to (-403.75, 334.43, 2.08) mm, rotated rx 180 ry 0 rz 0.01 deg; joints [35.411, -32.563, 74.924, -133.86, 53.502, 149.184]
  MoveL 793 to (-403.78, 333.95, 2.06) mm, rotated rx -180 ry 0 rz 0.01 deg; joints [35.398, -32.578, 74.956, -133.884, 53.507, 149.209]
  MoveL 794 to (-403.79, 333.65, 2.05) mm, rotated rx 180 ry 0 rz 0.01 deg; joints [35.39, -32.587, 74.977, -133.898, 53.511, 149.224]
  MoveL 795 to (-403.79, 333.05, 2.03) mm, rotated rx 180 ry 0 rz 0.01 deg; joints [35.374, -32.608, 75.021, -133.927, 53.519, 149.255]
  MoveL 796 to (-401.25, 328.08, 1.83) mm, rotated rx -180 ry 0 rz 0.01 deg; joints [35.29, -32.903, 75.645, -134.19, 53.703, 149.602]
  MoveL 797 to (-395.74, 327.2, 1.63) mm, rotated rx 180 ry 0 rz 0.01 deg; joints [35.371, -33.201, 76.271, -134.276, 53.974, 149.842]
  MoveL 798 to (-391.79, 331.15, 1.43) mm, rotated rx -180 ry 0 rz 0.01 deg; joints [35.551, -33.252, 76.386, -134.121, 54.112, 149.786]
  MoveL 799 to (-392.66, 336.66, 1.22) mm, rotated rx -180 ry 0 rz 0.01 deg; joints [35.68, -33.007, 75.896, -133.857, 54.011, 149.487]
  MoveL 800 to (-397.64, 339.2, 1.02) mm, rotated rx -180 ry 0 rz 0.01 deg; joints [35.653, -32.659, 75.201, -133.703, 53.756, 149.194]
  MoveL 801 to (-398.51, 339.2, 0.99) mm, rotated rx -180 ry 0 rz 0.01 deg; joints [35.636, -32.614, 75.112, -133.697, 53.717, 149.164]
  MoveL 802 to (-399.34, 339.13, 0.96) mm, rotated rx 180 ry 0 rz 0.01 deg; joints [35.619, -32.574, 75.031, -133.694, 53.68, 149.14]
  MoveL 803 to (-399.69, 339.08, 0.95) mm, rotated rx -180 ry 0 rz 0.01 deg; joints [35.611, -32.557, 74.999, -133.694, 53.664, 149.13]
  MoveL 804 to (-400.55, 338.85, 0.92) mm, rotated rx -180 ry 0 rz 0.01 deg; joints [35.589, -32.52, 74.927, -133.698, 53.628, 149.113]
  MoveL 805 to (-400.6, 338.83, 0.92) mm, rotated rx -180 ry 0 rz 0.01 deg; joints [35.587, -32.519, 74.923, -133.699, 53.626, 149.112]
  MoveL 806 to (-401.28, 338.49, 0.89) mm, rotated rx 180 ry 0 rz 0.01 deg; joints [35.566, -32.495, 74.877, -133.71, 53.6, 149.106]
  MoveL 807 to (-401.4, 338.42, 0.88) mm, rotated rx -180 ry 0 rz 0.01 deg; joints [35.561, -32.491, 74.87, -133.713, 53.595, 149.106]
  MoveL 808 to (-402.84, 337.05, 0.81) mm, rotated rx 180 ry 0 rz 0.01 deg; joints [35.498, -32.464, 74.822, -133.768, 53.547, 149.127]
  MoveL 809 to (-402.87, 337.02, 0.81) mm, rotated rx -180 ry 0 rz 0.01 deg; joints [35.497, -32.464, 74.822, -133.769, 53.546, 149.128]
  MoveL 810 to (-403.75, 334.43, 0.72) mm, rotated rx -180 ry 0 rz 0.01 deg; joints [35.412, -32.506, 74.921, -133.888, 53.54, 149.232]
  MoveL 811 to (-403.78, 333.95, 0.7) mm, rotated rx 180 ry 0 rz 0.01 deg; joints [35.399, -32.522, 74.954, -133.912, 53.545, 149.256]
  MoveL 812 to (-403.79, 333.65, 0.69) mm, rotated rx 180 ry 0 rz 0.01 deg; joints [35.391, -32.531, 74.975, -133.926, 53.549, 149.271]
  MoveL 813 to (-403.79, 333.05, 0.67) mm, rotated rx -180 ry 0 rz 0.01 deg; joints [35.375, -32.552, 75.019, -133.955, 53.557, 149.303]
  MoveL 814 to (-401.25, 328.08, 0.47) mm, rotated rx -180 ry 0 rz 0.01 deg; joints [35.291, -32.846, 75.642, -134.218, 53.741, 149.65]
  MoveL 815 to (-395.74, 327.2, 0.26) mm, rotated rx -180 ry 0 rz 0.01 deg; joints [35.372, -33.145, 76.268, -134.304, 54.012, 149.889]
  MoveL 816 to (-391.79, 331.15, 0.06) mm, rotated rx 180 ry 0 rz 0.01 deg; joints [35.551, -33.195, 76.383, -134.148, 54.15, 149.833]
  MoveL 817 to (-392.66, 336.66, -0.14) mm, rotated rx -180 ry 0 rz 0.01 deg; joints [35.681, -32.951, 75.893, -133.885, 54.048, 149.535]
  MoveL 818 to (-397.64, 339.2, -0.34) mm, rotated rx -180 ry 0 rz 0.01 deg; joints [35.653, -32.603, 75.198, -133.731, 53.793, 149.241]
  MoveL 819 to (-398.51, 339.2, -0.37) mm, rotated rx -180 ry 0 rz 0.01 deg; joints [35.637, -32.558, 75.109, -133.724, 53.754, 149.212]
  MoveL 820 to (-399.34, 339.13, -0.4) mm, rotated rx -180 ry 0 rz 0.01 deg; joints [35.62, -32.517, 75.028, -133.722, 53.717, 149.187]
  MoveL 821 to (-399.69, 339.08, -0.42) mm, rotated rx 180 ry 0 rz 0.01 deg; joints [35.611, -32.501, 74.996, -133.722, 53.702, 149.178]
  MoveL 822 to (-400.55, 338.85, -0.45) mm, rotated rx -180 ry 0 rz 0.01 deg; joints [35.589, -32.464, 74.924, -133.726, 53.666, 149.161]
  MoveL 823 to (-400.6, 338.83, -0.45) mm, rotated rx -180 ry 0 rz 0.01 deg; joints [35.588, -32.462, 74.921, -133.727, 53.664, 149.16]
  MoveL 824 to (-401.28, 338.49, -0.47) mm, rotated rx -180 ry 0 rz 0.01 deg; joints [35.566, -32.438, 74.875, -133.738, 53.637, 149.154]
  MoveL 825 to (-401.4, 338.42, -0.48) mm, rotated rx -180 ry 0 rz 0.01 deg; joints [35.562, -32.435, 74.868, -133.741, 53.632, 149.154]
  MoveL 826 to (-402.84, 337.05, -0.55) mm, rotated rx -180 ry 0 rz 0.01 deg; joints [35.499, -32.407, 74.82, -133.796, 53.584, 149.175]
  MoveL 827 to (-402.87, 337.02, -0.55) mm, rotated rx -180 ry 0 rz 0.01 deg; joints [35.497, -32.407, 74.82, -133.797, 53.584, 149.176]
  MoveL 828 to (-403.75, 334.43, -0.65) mm, rotated rx 180 ry 0 rz 0.01 deg; joints [35.413, -32.45, 74.918, -133.916, 53.577, 149.28]
  MoveL 829 to (-403.78, 333.95, -0.66) mm, rotated rx 180 ry 0 rz 0.01 deg; joints [35.399, -32.465, 74.951, -133.94, 53.583, 149.304]
  MoveL 830 to (-403.79, 333.65, -0.68) mm, rotated rx -180 ry 0 rz 0.01 deg; joints [35.392, -32.475, 74.972, -133.954, 53.586, 149.319]
  MoveL 831 to (-403.79, 333.05, -0.7) mm, rotated rx -180 ry 0 rz 0.01 deg; joints [35.376, -32.495, 75.016, -133.983, 53.594, 149.351]
  MoveL 832 to (-401.25, 328.08, -0.9) mm, rotated rx -180 ry 0 rz 0.01 deg; joints [35.292, -32.79, 75.64, -134.245, 53.779, 149.697]
  MoveL 833 to (-395.74, 327.2, -1.1) mm, rotated rx 180 ry 0 rz 0.01 deg; joints [35.372, -33.088, 76.266, -134.331, 54.05, 149.937]
  MoveL 834 to (-391.79, 331.15, -1.3) mm, rotated rx -180 ry 0 rz 0.01 deg; joints [35.552, -33.139, 76.381, -134.176, 54.188, 149.881]
  MoveL 835 to (-392.66, 336.66, -1.51) mm, rotated rx -180 ry 0 rz 0.01 deg; joints [35.681, -32.894, 75.891, -133.912, 54.086, 149.582]
  MoveL 836 to (-397.64, 339.2, -1.71) mm, rotated rx 180 ry 0 rz 0.01 deg; joints [35.654, -32.546, 75.196, -133.758, 53.831, 149.289]
  MoveL 837 to (-398.51, 339.2, -1.74) mm, rotated rx -180 ry 0 rz 0.01 deg; joints [35.638, -32.501, 75.106, -133.752, 53.791, 149.26]
  MoveL 838 to (-399.34, 339.13, -1.77) mm, rotated rx -180 ry 0 rz 0.01 deg; joints [35.62, -32.461, 75.026, -133.749, 53.755, 149.235]
  MoveL 839 to (-399.69, 339.08, -1.78) mm, rotated rx -180 ry 0 rz 0.01 deg; joints [35.612, -32.444, 74.993, -133.75, 53.739, 149.226]
  MoveL 840 to (-400.55, 338.85, -1.81) mm, rotated rx -180 ry 0 rz 0.01 deg; joints [35.59, -32.407, 74.921, -133.754, 53.703, 149.208]
  MoveL 841 to (-400.6, 338.83, -1.81) mm, rotated rx -180 ry 0 rz 0.01 deg; joints [35.589, -32.406, 74.918, -133.755, 53.701, 149.208]
  MoveL 842 to (-401.28, 338.49, -1.84) mm, rotated rx 180 ry 0 rz 0.01 deg; joints [35.567, -32.382, 74.872, -133.766, 53.674, 149.202]
  MoveL 843 to (-401.4, 338.42, -1.84) mm, rotated rx -180 ry 0 rz 0.01 deg; joints [35.562, -32.378, 74.865, -133.769, 53.67, 149.201]
  MoveL 844 to (-402.84, 337.05, -1.91) mm, rotated rx -180 ry 0 rz 0.01 deg; joints [35.499, -32.351, 74.817, -133.824, 53.622, 149.223]
  MoveL 845 to (-402.87, 337.02, -1.92) mm, rotated rx 180 ry 0 rz 0.01 deg; joints [35.498, -32.351, 74.817, -133.825, 53.621, 149.224]
  MoveL 846 to (-403.75, 334.43, -2.01) mm, rotated rx 180 ry 0 rz 0.01 deg; joints [35.413, -32.394, 74.915, -133.944, 53.615, 149.327]
  MoveL 847 to (-403.78, 333.95, -2.03) mm, rotated rx -180 ry 0 rz 0.01 deg; joints [35.4, -32.409, 74.948, -133.967, 53.62, 149.352]
  MoveL 848 to (-403.79, 333.65, -2.04) mm, rotated rx -180 ry 0 rz 0.01 deg; joints [35.392, -32.418, 74.969, -133.982, 53.624, 149.367]
  MoveL 849 to (-403.79, 333.05, -2.06) mm, rotated rx -180 ry 0 rz 0.01 deg; joints [35.376, -32.439, 75.013, -134.011, 53.632, 149.398]
  MoveL 850 to (-401.25, 328.08, -2.26) mm, rotated rx -180 ry 0 rz 0.01 deg; joints [35.292, -32.733, 75.637, -134.273, 53.817, 149.745]
  MoveL 851 to (-395.74, 327.2, -2.47) mm, rotated rx -180 ry 0 rz 0.01 deg; joints [35.373, -33.031, 76.263, -134.359, 54.088, 149.984]
  MoveL 852 to (-391.79, 331.15, -2.67) mm, rotated rx 180 ry 0 rz 0.01 deg; joints [35.552, -33.082, 76.378, -134.203, 54.226, 149.928]
  MoveL 853 to (-392.66, 336.66, -2.87) mm, rotated rx 180 ry 0 rz 0.01 deg; joints [35.682, -32.837, 75.888, -133.94, 54.124, 149.63]
  MoveL 854 to (-397.64, 339.2, -3.07) mm, rotated rx -180 ry 0 rz 0.01 deg; joints [35.654, -32.49, 75.193, -133.786, 53.868, 149.337]
  MoveL 855 to (-398.51, 339.2, -3.1) mm, rotated rx -180 ry 0 rz 0.01 deg; joints [35.638, -32.445, 75.103, -133.78, 53.829, 149.307]
  MoveL 856 to (-399.34, 339.13, -3.13) mm, rotated rx -180 ry 0 rz 0.01 deg; joints [35.621, -32.404, 75.023, -133.777, 53.792, 149.283]
  MoveL 857 to (-399.69, 339.08, -3.14) mm, rotated rx 180 ry 0 rz 0.01 deg; joints [35.613, -32.388, 74.99, -133.777, 53.776, 149.273]
  MoveL 858 to (-400.55, 338.85, -3.18) mm, rotated rx -180 ry 0 rz 0.01 deg; joints [35.59, -32.351, 74.918, -133.782, 53.74, 149.256]
  MoveL 859 to (-400.6, 338.83, -3.18) mm, rotated rx -180 ry 0 rz 0.01 deg; joints [35.589, -32.349, 74.915, -133.782, 53.738, 149.255]
  MoveL 860 to (-401.28, 338.49, -3.2) mm, rotated rx -180 ry 0 rz 0.01 deg; joints [35.567, -32.325, 74.869, -133.794, 53.712, 149.249]
  MoveL 861 to (-401.4, 338.42, -3.21) mm, rotated rx -180 ry 0 rz 0.01 deg; joints [35.563, -32.322, 74.862, -133.796, 53.707, 149.249]
  MoveL 862 to (-402.84, 337.05, -3.28) mm, rotated rx -180 ry 0 rz 0.01 deg; joints [35.5, -32.294, 74.814, -133.851, 53.659, 149.27]
  MoveL 863 to (-402.87, 337.02, -3.28) mm, rotated rx -180 ry 0 rz 0.01 deg; joints [35.499, -32.294, 74.814, -133.853, 53.658, 149.271]
  MoveL 864 to (-403.75, 334.43, -3.38) mm, rotated rx -180 ry 0 rz 0.01 deg; joints [35.414, -32.337, 74.912, -133.972, 53.652, 149.375]
  MoveL 865 to (-403.78, 333.95, -3.39) mm, rotated rx -180 ry 0 rz 0.01 deg; joints [35.401, -32.352, 74.945, -133.995, 53.658, 149.399]
  MoveL 866 to (-403.79, 333.65, -3.4) mm, rotated rx 180 ry 0 rz 0.01 deg; joints [35.393, -32.362, 74.966, -134.009, 53.661, 149.414]
  MoveL 867 to (-403.79, 333.05, -3.43) mm, rotated rx 180 ry 0 rz 0.01 deg; joints [35.377, -32.382, 75.01, -134.039, 53.669, 149.445]
  MoveL 868 to (-401.25, 328.08, -3.63) mm, rotated rx -180 ry 0 rz 0.01 deg; joints [35.293, -32.676, 75.634, -134.3, 53.855, 149.792]
  MoveL 869 to (-395.74, 327.2, -3.83) mm, rotated rx -180 ry 0 rz 0.01 deg; joints [35.373, -32.974, 76.26, -134.386, 54.126, 150.031]
  MoveL 870 to (-391.79, 331.15, -4.03) mm, rotated rx -180 ry 0 rz 0.01 deg; joints [35.553, -33.025, 76.375, -134.23, 54.264, 149.975]
  MoveL 871 to (-392.66, 336.66, -4.23) mm, rotated rx 180 ry 0 rz 0.01 deg; joints [35.682, -32.78, 75.885, -133.967, 54.161, 149.677]
  MoveL 872 to (-397.64, 339.2, -4.44) mm, rotated rx 180 ry 0 rz 0.01 deg; joints [35.655, -32.433, 75.189, -133.814, 53.905, 149.384]
  MoveL 873 to (-398.51, 339.2, -4.47) mm, rotated rx 180 ry 0 rz 0.01 deg; joints [35.639, -32.388, 75.1, -133.808, 53.866, 149.355]
  MoveL 874 to (-399.34, 339.13, -4.5) mm, rotated rx -180 ry 0 rz 0.01 deg; joints [35.621, -32.347, 75.019, -133.805, 53.829, 149.33]
  MoveL 875 to (-399.69, 339.08, -4.51) mm, rotated rx 180 ry 0 rz 0.01 deg; joints [35.613, -32.331, 74.987, -133.805, 53.814, 149.321]
  MoveL 876 to (-400.55, 338.85, -4.54) mm, rotated rx -180 ry 0 rz 0.01 deg; joints [35.591, -32.294, 74.915, -133.81, 53.778, 149.303]
  MoveL 877 to (-400.6, 338.83, -4.54) mm, rotated rx -180 ry 0 rz 0.01 deg; joints [35.59, -32.293, 74.912, -133.81, 53.776, 149.303]
  MoveL 878 to (-401.28, 338.49, -4.57) mm, rotated rx -180 ry 0 rz 0.01 deg; joints [35.568, -32.269, 74.866, -133.821, 53.749, 149.297]
  MoveL 879 to (-401.4, 338.42, -4.57) mm, rotated rx -180 ry 0 rz 0.01 deg; joints [35.564, -32.265, 74.859, -133.824, 53.744, 149.296]
  MoveL 880 to (-402.84, 337.05, -4.64) mm, rotated rx 180 ry 0 rz 0.01 deg; joints [35.501, -32.238, 74.81, -133.879, 53.696, 149.318]
  MoveL 881 to (-402.87, 337.02, -4.64) mm, rotated rx -180 ry 0 rz 0.01 deg; joints [35.499, -32.238, 74.811, -133.881, 53.696, 149.318]
  MoveL 882 to (-403.75, 334.43, -4.74) mm, rotated rx -180 ry 0 rz 0.01 deg; joints [35.414, -32.28, 74.909, -133.999, 53.69, 149.422]
  MoveL 883 to (-403.78, 333.95, -4.76) mm, rotated rx -180 ry 0 rz 0.01 deg; joints [35.401, -32.296, 74.942, -134.023, 53.695, 149.446]
  MoveL 884 to (-403.79, 333.65, -4.77) mm, rotated rx -180 ry 0 rz 0.01 deg; joints [35.393, -32.305, 74.963, -134.037, 53.699, 149.461]
  MoveL 885 to (-403.79, 333.05, -4.79) mm, rotated rx -180 ry 0 rz 0.01 deg; joints [35.377, -32.325, 75.007, -134.066, 53.707, 149.493]
  MoveL 886 to (-401.25, 328.08, -4.99) mm, rotated rx 180 ry 0 rz 0.01 deg; joints [35.293, -32.619, 75.631, -134.328, 53.892, 149.839]
  MoveL 887 to (-395.74, 327.2, -5.19) mm, rotated rx -180 ry 0 rz 0.01 deg; joints [35.374, -32.917, 76.256, -134.413, 54.164, 150.078]
  MoveL 888 to (-391.79, 331.15, -5.4) mm, rotated rx -180 ry 0 rz 0.01 deg; joints [35.553, -32.968, 76.371, -134.257, 54.302, 150.022]
  MoveL 889 to (-392.66, 336.66, -5.6) mm, rotated rx -180 ry 0 rz 0.01 deg; joints [35.683, -32.723, 75.881, -133.994, 54.199, 149.724]
  MoveL 890 to (-397.64, 339.2, -5.8) mm, rotated rx 180 ry 0 rz 0.01 deg; joints [35.656, -32.376, 75.186, -133.841, 53.943, 149.431]
  MoveL 891 to (-398.51, 339.2, -5.83) mm, rotated rx 180 ry 0 rz 0.01 deg; joints [35.639, -32.331, 75.097, -133.835, 53.903, 149.402]
  MoveL 892 to (-399.34, 339.13, -5.86) mm, rotated rx -180 ry 0 rz 0.01 deg; joints [35.622, -32.291, 75.016, -133.832, 53.867, 149.377]
  MoveL 893 to (-399.69, 339.08, -5.87) mm, rotated rx -180 ry 0 rz 0.01 deg; joints [35.614, -32.274, 74.983, -133.832, 53.851, 149.368]
  MoveL 894 to (-400.55, 338.85, -5.9) mm, rotated rx -180 ry 0 rz 0.01 deg; joints [35.592, -32.238, 74.912, -133.837, 53.815, 149.351]
  MoveL 895 to (-400.6, 338.83, -5.91) mm, rotated rx -180 ry 0 rz 0.01 deg; joints [35.59, -32.236, 74.908, -133.838, 53.813, 149.35]
  MoveL 896 to (-401.28, 338.49, -5.93) mm, rotated rx 180 ry 0 rz 0.01 deg; joints [35.568, -32.212, 74.862, -133.849, 53.786, 149.344]
  MoveL 897 to (-401.4, 338.42, -5.94) mm, rotated rx 180 ry 0 rz 0.01 deg; joints [35.564, -32.208, 74.855, -133.852, 53.782, 149.344]
  MoveL 898 to (-402.84, 337.05, -6.01) mm, rotated rx -180 ry 0 rz 0.01 deg; joints [35.501, -32.181, 74.807, -133.907, 53.734, 149.365]
  MoveL 899 to (-402.87, 337.02, -6.01) mm, rotated rx -180 ry 0 rz 0.01 deg; joints [35.5, -32.181, 74.807, -133.908, 53.733, 149.366]
  MoveL 900 to (-403.75, 334.43, -6.11) mm, rotated rx -180 ry 0 rz 0.01 deg; joints [35.415, -32.224, 74.906, -134.027, 53.727, 149.469]
  MoveL 901 to (-403.78, 333.95, -6.12) mm, rotated rx -180 ry 0 rz 0.01 deg; joints [35.402, -32.239, 74.939, -134.05, 53.732, 149.494]
  MoveL 902 to (-403.79, 333.65, -6.13) mm, rotated rx -180 ry 0 rz 0.01 deg; joints [35.394, -32.248, 74.959, -134.064, 53.736, 149.509]
  MoveL 903 to (-403.79, 333.05, -6.15) mm, rotated rx 180 ry 0 rz 0.01 deg; joints [35.378, -32.269, 75.004, -134.094, 53.744, 149.54]
  MoveL 904 to (-401.25, 328.08, -6.36) mm, rotated rx 180 ry 0 rz 0.01 deg; joints [35.294, -32.562, 75.627, -134.355, 53.93, 149.886]
  MoveL 905 to (-395.74, 327.2, -6.56) mm, rotated rx 180 ry 0 rz 0.01 deg; joints [35.375, -32.86, 76.253, -134.44, 54.202, 150.125]
  MoveL 906 to (-391.79, 331.15, -6.76) mm, rotated rx -180 ry 0 rz 0.01 deg; joints [35.554, -32.91, 76.368, -134.284, 54.34, 150.069]
  MoveL 907 to (-392.66, 336.66, -6.96) mm, rotated rx -180 ry 0 rz 0.01 deg; joints [35.683, -32.666, 75.878, -134.022, 54.236, 149.771]
  MoveL 908 to (-397.64, 339.2, -7.17) mm, rotated rx -180 ry 0 rz 0.01 deg; joints [35.656, -32.32, 75.183, -133.869, 53.98, 149.479]
  MoveL 909 to (-398.51, 339.2, -7.2) mm, rotated rx -180 ry 0 rz 0.01 deg; joints [35.64, -32.275, 75.093, -133.862, 53.941, 149.449]
  MoveL 910 to (-399.34, 339.13, -7.23) mm, rotated rx -180 ry 0 rz 0.01 deg; joints [35.623, -32.234, 75.013, -133.86, 53.904, 149.425]
  MoveL 911 to (-399.69, 339.08, -7.24) mm, rotated rx 180 ry 0 rz 0.01 deg; joints [35.614, -32.217, 74.98, -133.86, 53.888, 149.415]
  MoveL 912 to (-400.55, 338.85, -7.27) mm, rotated rx -180 ry 0 rz 0.01 deg; joints [35.592, -32.181, 74.908, -133.865, 53.852, 149.398]
  MoveL 913 to (-400.6, 338.83, -7.27) mm, rotated rx -180 ry 0 rz 0.01 deg; joints [35.591, -32.179, 74.905, -133.865, 53.85, 149.397]
  MoveL 914 to (-401.28, 338.49, -7.3) mm, rotated rx 180 ry 0 rz 0.01 deg; joints [35.569, -32.155, 74.859, -133.876, 53.823, 149.391]
  MoveL 915 to (-401.4, 338.42, -7.3) mm, rotated rx 180 ry 0 rz 0.01 deg; joints [35.565, -32.152, 74.852, -133.879, 53.819, 149.391]
  MoveL 916 to (-402.84, 337.05, -7.37) mm, rotated rx -180 ry 0 rz 0.01 deg; joints [35.502, -32.124, 74.804, -133.934, 53.771, 149.412]
  MoveL 917 to (-402.87, 337.02, -7.37) mm, rotated rx -180 ry 0 rz 0.01 deg; joints [35.5, -32.124, 74.804, -133.936, 53.77, 149.413]
  MoveL 918 to (-403.75, 334.43, -7.47) mm, rotated rx 180 ry 0 rz 0.01 deg; joints [35.416, -32.167, 74.902, -134.054, 53.764, 149.516]
  MoveL 919 to (-403.78, 333.95, -7.49) mm, rotated rx -180 ry 0 rz 0.01 deg; joints [35.402, -32.182, 74.935, -134.078, 53.77, 149.541]
  MoveL 920 to (-403.79, 333.65, -7.5) mm, rotated rx -180 ry 0 rz 0.01 deg; joints [35.395, -32.192, 74.956, -134.092, 53.773, 149.556]
  MoveL 921 to (-403.79, 333.05, -7.52) mm, rotated rx -180 ry 0 rz 0.01 deg; joints [35.379, -32.212, 75, -134.121, 53.782, 149.587]
  MoveL 922 to (-401.25, 328.08, -7.72) mm, rotated rx -180 ry 0 rz 0.01 deg; joints [35.295, -32.505, 75.624, -134.382, 53.968, 149.933]
  MoveL 923 to (-395.74, 327.2, -7.92) mm, rotated rx 180 ry 0 rz 0.01 deg; joints [35.375, -32.803, 76.249, -134.467, 54.24, 150.172]
  MoveL 924 to (-391.79, 331.15, -8.13) mm, rotated rx -180 ry 0 rz 0.01 deg; joints [35.555, -32.853, 76.364, -134.311, 54.378, 150.116]
  MoveL 925 to (-392.66, 336.66, -8.33) mm, rotated rx 180 ry 0 rz 0.01 deg; joints [35.684, -32.609, 75.874, -134.049, 54.274, 149.818]
  MoveL 926 to (-397.64, 339.2, -8.53) mm, rotated rx -180 ry 0 rz 0.01 deg; joints [35.657, -32.263, 75.179, -133.896, 54.017, 149.526]
  MoveL 927 to (-398.51, 339.2, -8.56) mm, rotated rx 180 ry 0 rz 0.01 deg; joints [35.64, -32.218, 75.089, -133.89, 53.978, 149.496]
  MoveL 928 to (-399.34, 339.13, -8.59) mm, rotated rx 180 ry 0 rz 0.01 deg; joints [35.623, -32.177, 75.009, -133.887, 53.941, 149.472]
  MoveL 929 to (-399.69, 339.08, -8.6) mm, rotated rx -180 ry 0 rz 0.01 deg; joints [35.615, -32.161, 74.976, -133.887, 53.925, 149.462]
  MoveL 930 to (-400.55, 338.85, -8.63) mm, rotated rx -180 ry 0 rz 0.01 deg; joints [35.593, -32.124, 74.904, -133.892, 53.889, 149.445]
  MoveL 931 to (-400.6, 338.83, -8.64) mm, rotated rx -180 ry 0 rz 0.01 deg; joints [35.591, -32.122, 74.901, -133.892, 53.887, 149.444]
  MoveL 932 to (-401.28, 338.49, -8.66) mm, rotated rx -180 ry 0 rz 0.01 deg; joints [35.57, -32.099, 74.855, -133.904, 53.86, 149.438]
  MoveL 933 to (-401.4, 338.42, -8.67) mm, rotated rx -180 ry 0 rz 0.01 deg; joints [35.565, -32.095, 74.848, -133.906, 53.856, 149.438]
  MoveL 934 to (-402.84, 337.05, -8.74) mm, rotated rx -180 ry 0 rz 0.01 deg; joints [35.502, -32.068, 74.8, -133.961, 53.808, 149.459]
  MoveL 935 to (-402.87, 337.02, -8.74) mm, rotated rx -180 ry 0 rz 0.01 deg; joints [35.501, -32.068, 74.8, -133.963, 53.807, 149.46]
  MoveL 936 to (-403.75, 334.43, -8.84) mm, rotated rx 180 ry 0 rz 0.01 deg; joints [35.416, -32.11, 74.898, -134.082, 53.802, 149.563]
  MoveL 937 to (-403.78, 333.95, -8.85) mm, rotated rx -180 ry 0 rz 0.01 deg; joints [35.403, -32.125, 74.931, -134.105, 53.807, 149.588]
  MoveL 938 to (-403.79, 333.65, -8.86) mm, rotated rx -180 ry 0 rz 0.01 deg; joints [35.395, -32.135, 74.952, -134.119, 53.811, 149.603]
  MoveL 939 to (-403.79, 333.05, -8.88) mm, rotated rx -180 ry 0 rz 0.01 deg; joints [35.379, -32.155, 74.996, -134.148, 53.819, 149.634]
  MoveL 940 to (-401.25, 328.08, -9.09) mm, rotated rx 180 ry 0 rz 0.01 deg; joints [35.295, -32.448, 75.62, -134.409, 54.006, 149.98]
  MoveL 941 to (-395.74, 327.2, -9.29) mm, rotated rx 180 ry 0 rz 0.01 deg; joints [35.376, -32.745, 76.246, -134.494, 54.278, 150.219]
  MoveL 942 to (-391.79, 331.15, -9.49) mm, rotated rx -180 ry 0 rz 0.01 deg; joints [35.555, -32.796, 76.36, -134.338, 54.416, 150.163]
  MoveL 943 to (-392.66, 336.66, -9.69) mm, rotated rx 180 ry 0 rz 0.01 deg; joints [35.685, -32.552, 75.87, -134.076, 54.311, 149.865]
  MoveL 944 to (-397.64, 339.2, -9.9) mm, rotated rx -180 ry 0 rz 0.01 deg; joints [35.657, -32.206, 75.175, -133.923, 54.054, 149.573]
  MoveL 945 to (-398.51, 339.2, -9.93) mm, rotated rx -180 ry 0 rz 0.01 deg; joints [35.641, -32.161, 75.086, -133.917, 54.015, 149.543]
  MoveL 946 to (-399.34, 339.13, -9.95) mm, rotated rx -180 ry 0 rz 0.01 deg; joints [35.624, -32.12, 75.005, -133.914, 53.978, 149.519]
  MoveL 947 to (-399.69, 339.08, -9.97) mm, rotated rx -180 ry 0 rz 0.01 deg; joints [35.615, -32.104, 74.972, -133.914, 53.963, 149.509]
  MoveL 948 to (-400.55, 338.85, -10) mm, rotated rx 180 ry 0 rz 0.01 deg; joints [35.593, -32.067, 74.9, -133.919, 53.926, 149.492]
  MoveL 949 to (-400.6, 338.83, -10) mm, rotated rx -180 ry 0 rz 0.01 deg; joints [35.592, -32.065, 74.897, -133.92, 53.925, 149.491]
  MoveL 950 to (-400.13, 339.01, -10) mm, rotated rx -180 ry 0 rz 0.01 deg; joints [35.605, -32.083, 74.932, -133.915, 53.944, 149.499]
  MoveL 951 to (-398.92, 339.2, -10) mm, rotated rx 180 ry 0 rz 0.01 deg; joints [35.633, -32.137, 75.042, -133.915, 53.998, 149.531]
  MoveL 952 to (-213.12, 339.2, -10) mm, rotated rx 180 ry 0 rz 0.01 deg; joints [39.46, -40.316, 91.85, -133.868, 61.858, 154.734]
  MoveL 953 to (-213.23, 339.19, -10) mm, rotated rx -180 ry 0 rz 0.01 deg; joints [39.458, -40.312, 91.843, -133.87, 61.854, 154.732]
  MoveL 954 to (-213.44, 339.15, -10) mm, rotated rx -180 ry 0 rz 0.01 deg; joints [39.452, -40.305, 91.829, -133.873, 61.847, 154.729]
  MoveL 955 to (-214.53, 338.91, -10) mm, rotated rx 180 ry 0 rz 0.01 deg; joints [39.421, -40.27, 91.757, -133.89, 61.807, 154.714]
  MoveL 956 to (-215.3, 338.64, -10) mm, rotated rx 180 ry 0 rz 0.01 deg; joints [39.396, -40.248, 91.712, -133.906, 61.78, 154.708]
  MoveL 957 to (-225.82, 333.47, -10) mm, rotated rx -180 ry 0 rz 0.01 deg; joints [39.02, -39.998, 91.203, -134.187, 61.431, 154.682]
  MoveL 958 to (-226, 333.37, -10) mm, rotated rx 180 ry 0 rz 0.01 deg; joints [39.014, -39.994, 91.194, -134.192, 61.426, 154.681]
  MoveL 959 to (-227.45, 332.55, -10) mm, rotated rx 180 ry 0 rz 0.01 deg; joints [38.959, -39.962, 91.131, -134.235, 61.378, 154.682]
  MoveL 960 to (-228.12, 332.04, -10) mm, rotated rx -180 ry 0 rz 0.01 deg; joints [38.931, -39.951, 91.109, -134.26, 61.358, 154.688]
  MoveL 961 to (-237.25, 323.27, -10) mm, rotated rx 180 ry 0 rz 0.01 deg; joints [38.489, -39.862, 90.937, -134.678, 61.103, 154.842]
  MoveL 962 to (-237.62, 322.85, -10) mm, rotated rx 180 ry 0 rz 0.01 deg; joints [38.47, -39.861, 90.934, -134.697, 61.093, 154.851]
  MoveL 963 to (-238.16, 322.12, -10) mm, rotated rx 180 ry 0 rz 0.01 deg; joints [38.438, -39.862, 90.937, -134.73, 61.08, 154.869]
  MoveL 964 to (-238.41, 321.72, -10) mm, rotated rx -180 ry 0 rz 0.01 deg; joints [38.421, -39.864, 90.943, -134.749, 61.075, 154.879]
  MoveL 965 to (-243.93, 311.56, -10) mm, rotated rx 180 ry 0 rz 0.01 deg; joints [38.02, -39.956, 91.147, -135.203, 60.976, 155.173]
  MoveL 966 to (-244.05, 311.32, -10) mm, rotated rx 180 ry 0 rz 0.01 deg; joints [38.011, -39.958, 91.152, -135.214, 60.974, 155.181]
  MoveL 967 to (-244.69, 309.87, -10) mm, rotated rx 180 ry 0 rz 0.01 deg; joints [37.957, -39.977, 91.193, -135.278, 60.966, 155.226]
  MoveL 968 to (-244.95, 309.01, -10) mm, rotated rx 180 ry 0 rz 0.01 deg; joints [37.928, -39.993, 91.227, -135.315, 60.966, 155.255]
  MoveL 969 to (-246.39, 299.58, -10) mm, rotated rx 180 ry 0 rz 0.01 deg; joints [37.634, -40.22, 91.711, -135.717, 61.02, 155.61]
  MoveL 970 to (-246.42, 299.36, -10) mm, rotated rx 180 ry 0 rz 0.01 deg; joints [37.627, -40.226, 91.723, -135.726, 61.022, 155.619]
  MoveL 971 to (-246.51, 298.27, -10) mm, rotated rx 180 ry 0 rz 0.01 deg; joints [37.595, -40.255, 91.784, -135.772, 61.031, 155.661]
  MoveC 972 to (-246.51, 297.75, -10) mm, rotated rx -180 ry 0 rz 0.01 deg; joints [37.58, -40.27, 91.817, -135.794, 61.037, 155.682] to (-246.44, 297.23, -10) mm, rotated rx -180 ry 0 rz 0.01 deg; joints [37.567, -40.289, 91.856, -135.815, 61.046, 155.705]
  MoveL 973 to (-245.04, 291.06, -10) mm, rotated rx 180 ry 0 rz 0.01 deg; joints [37.424, -40.529, 92.36, -136.064, 61.175, 155.988]
  MoveL 974 to (-245.03, 291.01, -10) mm, rotated rx -180 ry 0 rz 0.01 deg; joints [37.423, -40.531, 92.364, -136.066, 61.176, 155.99]
  MoveL 975 to (-244.06, 287.02, -10) mm, rotated rx 180 ry 0 rz 0.01 deg; joints [37.331, -40.687, 92.693, -136.226, 61.261, 156.173]
  MoveL 976 to (-243.78, 286.27, -10) mm, rotated rx -180 ry 0 rz 0.01 deg; joints [37.316, -40.721, 92.764, -136.256, 61.281, 156.21]
  MoveL 977 to (-243.05, 284.86, -10) mm, rotated rx -180 ry 0 rz 0.01 deg; joints [37.292, -40.791, 92.912, -136.31, 61.327, 156.283]
  MoveL 978 to (-242.81, 284.46, -10) mm, rotated rx 180 ry 0 rz 0.01 deg; joints [37.286, -40.812, 92.955, -136.325, 61.341, 156.304]
  MoveL 979 to (-238.71, 278.61, -10) mm, rotated rx -180 ry 0 rz 0.01 deg; joints [37.208, -41.146, 93.654, -136.542, 61.572, 156.63]
  MoveL 980 to (-238.58, 278.44, -10) mm, rotated rx 180 ry 0 rz 0.01 deg; joints [37.206, -41.156, 93.675, -136.548, 61.579, 156.639]
  MoveL 981 to (-237.13, 276.64, -10) mm, rotated rx -180 ry 0 rz 0.01 deg; joints [37.186, -41.265, 93.903, -136.613, 61.658, 156.742]
  MoveL 982 to (-236.64, 276.14, -10) mm, rotated rx -180 ry 0 rz 0.01 deg; joints [37.183, -41.299, 93.974, -136.63, 61.683, 156.773]
  MoveL 983 to (-235.91, 275.54, -10) mm, rotated rx -180 ry 0 rz 0.01 deg; joints [37.181, -41.344, 94.07, -136.65, 61.719, 156.813]
  MoveL 984 to (-235.62, 275.33, -10) mm, rotated rx 180 ry 0 rz 0.01 deg; joints [37.182, -41.362, 94.106, -136.657, 61.733, 156.827]
  MoveL 985 to (-229.09, 271.02, -10) mm, rotated rx -180 ry 0 rz 0.01 deg; joints [37.2, -41.741, 94.896, -136.788, 62.04, 157.138]
  MoveL 986 to (-228.91, 270.91, -10) mm, rotated rx -180 ry 0 rz 0.01 deg; joints [37.201, -41.751, 94.918, -136.792, 62.049, 157.146]
  MoveL 987 to (-227.33, 270.01, -10) mm, rotated rx -180 ry 0 rz 0.01 deg; joints [37.209, -41.838, 95.1, -136.817, 62.121, 157.215]
  MoveL 988 to (-226.81, 269.77, -10) mm, rotated rx -180 ry 0 rz 0.01 deg; joints [37.214, -41.865, 95.156, -136.823, 62.144, 157.236]
  MoveL 989 to (-225.49, 269.29, -10) mm, rotated rx 180 ry 0 rz 0.01 deg; joints [37.229, -41.93, 95.291, -136.833, 62.201, 157.283]
  MoveL 990 to (-224.98, 269.14, -10) mm, rotated rx 180 ry 0 rz 0.01 deg; joints [37.236, -41.954, 95.341, -136.835, 62.223, 157.299]
  MoveL 991 to (-219.17, 268.01, -10) mm, rotated rx 180 ry 0 rz 0.01 deg; joints [37.33, -42.21, 95.873, -136.837, 62.463, 157.466]
  MoveL 992 to (-219.06, 267.99, -10) mm, rotated rx 180 ry 0 rz 0.01 deg; joints [37.332, -42.215, 95.884, -136.837, 62.468, 157.469]
  MoveL 993 to (-215.43, 267.41, -10) mm, rotated rx 180 ry 0 rz 0.01 deg; joints [37.395, -42.371, 96.206, -136.831, 62.615, 157.568]
  MoveL 994 to (-214.9, 267.36, -10) mm, rotated rx 180 ry 0 rz 0.01 deg; joints [37.406, -42.392, 96.251, -136.829, 62.636, 157.581]
  MoveL 995 to (-179.34, 267.36, -10) mm, rotated rx -180 ry 0 rz 0.01 deg; joints [38.204, -43.725, 99.015, -136.503, 63.995, 158.304]
  MoveL 996 to (-179.13, 267.37, -10) mm, rotated rx 180 ry 0 rz 0.01 deg; joints [38.209, -43.732, 99.031, -136.501, 64.003, 158.308]
  MoveL 997 to (-177.68, 267.45, -10) mm, rotated rx 180 ry 0 rz 0.01 deg; joints [38.245, -43.783, 99.136, -136.482, 64.057, 158.333]
  MoveL 998 to (-177.28, 267.5, -10) mm, rotated rx 180 ry 0 rz 0.01 deg; joints [38.255, -43.797, 99.164, -136.476, 64.071, 158.339]
  MoveL 999 to (-169.29, 268.98, -10) mm, rotated rx -180 ry 0 rz 0.01 deg; joints [38.482, -44.047, 99.681, -136.334, 64.353, 158.44]
  MoveL 1000 to (-169.03, 269.04, -10) mm, rotated rx -180 ry 0 rz 0.01 deg; joints [38.49, -44.054, 99.698, -136.328, 64.362, 158.443]
  MoveL 1001 to (-167.65, 269.41, -10) mm, rotated rx -180 ry 0 rz 0.01 deg; joints [38.533, -44.094, 99.78, -136.299, 64.41, 158.457]
  MoveL 1002 to (-167.18, 269.58, -10) mm, rotated rx 180 ry 0 rz 0.01 deg; joints [38.548, -44.107, 99.806, -136.287, 64.425, 158.46]
  MoveL 1003 to (-166.12, 270.03, -10) mm, rotated rx -180 ry 0 rz 0.01 deg; joints [38.586, -44.132, 99.858, -136.258, 64.459, 158.463]
  MoveL 1004 to (-165.64, 270.29, -10) mm, rotated rx 180 ry 0 rz 0.01 deg; joints [38.604, -44.142, 99.879, -136.242, 64.474, 158.463]
  MoveL 1005 to (-158.65, 274.77, -10) mm, rotated rx 180 ry 0 rz 0.01 deg; joints [38.897, -44.269, 100.134, -135.986, 64.681, 158.431]
  MoveL 1006 to (-158.46, 274.9, -10) mm, rotated rx -180 ry 0 rz 0.01 deg; joints [38.905, -44.272, 100.14, -135.979, 64.687, 158.429]
  MoveL 1007 to (-157.37, 275.71, -10) mm, rotated rx 180 ry 0 rz 0.01 deg; joints [38.954, -44.288, 100.173, -135.934, 64.718, 158.42]
  MoveL 1008 to (-156.91, 276.12, -10) mm, rotated rx 180 ry 0 rz 0.01 deg; joints [38.977, -44.293, 100.183, -135.913, 64.73, 158.414]
  MoveL 1009 to (-155.77, 277.35, -10) mm, rotated rx 180 ry 0 rz 0.01 deg; joints [39.039, -44.299, 100.194, -135.851, 64.758, 158.39]
  MoveL 1010 to (-155.49, 277.69, -10) mm, rotated rx 180 ry 0 rz 0.01 deg; joints [39.056, -44.3, 100.194, -135.834, 64.764, 158.382]
  MoveL 1011 to (-150.93, 284.1, -10) mm, rotated rx -180 ry 0 rz 0.01 deg; joints [39.348, -44.281, 100.145, -135.527, 64.857, 158.229]
  MoveL 1012 to (-150.7, 284.46, -10) mm, rotated rx 180 ry 0 rz 0.01 deg; joints [39.364, -44.278, 100.139, -135.51, 64.861, 158.22]
  MoveL 1013 to (-149.76, 286.22, -10) mm, rotated rx -180 ry 0 rz 0.01 deg; joints [39.437, -44.262, 100.102, -135.429, 64.875, 158.172]
  MoveL 1014 to (-149.44, 287.04, -10) mm, rotated rx -180 ry 0 rz 0.01 deg; joints [39.468, -44.249, 100.075, -135.393, 64.877, 158.147]
  MoveL 1015 to (-147.12, 296.83, -10) mm, rotated rx 180 ry 0 rz 0.01 deg; joints [39.803, -44.05, 99.646, -134.977, 64.847, 157.82]
  MoveL 1016 to (-147.03, 297.45, -10) mm, rotated rx 180 ry 0 rz 0.01 deg; joints [39.823, -44.035, 99.614, -134.951, 64.843, 157.798]
  MoveL 1017 to (-146.99, 298.17, -10) mm, rotated rx -180 ry 0 rz 0.01 deg; joints [39.844, -44.015, 99.572, -134.922, 64.836, 157.771]
  MoveL 1018 to (-147.03, 298.84, -10) mm, rotated rx -180 ry 0 rz 0.01 deg; joints [39.862, -43.995, 99.528, -134.896, 64.827, 157.745]
  MoveL 1019 to (-148.48, 308.63, -10) mm, rotated rx 180 ry 0 rz 0.01 deg; joints [40.105, -43.656, 98.81, -134.523, 64.658, 157.339]
  MoveL 1020 to (-148.61, 309.17, -10) mm, rotated rx -180 ry 0 rz 0.01 deg; joints [40.118, -43.635, 98.767, -134.503, 64.647, 157.316]
  MoveL 1021 to (-148.96, 310.26, -10) mm, rotated rx 180 ry 0 rz 0.01 deg; joints [40.14, -43.591, 98.672, -134.464, 64.621, 157.266]
  MoveL 1022 to (-149.2, 310.83, -10) mm, rotated rx 180 ry 0 rz 0.01 deg; joints [40.15, -43.565, 98.618, -134.444, 64.605, 157.239]
  MoveL 1023 to (-155.09, 321.72, -10) mm, rotated rx 180 ry 0 rz 0.01 deg; joints [40.316, -43.028, 97.489, -134.074, 64.26, 156.695]
  MoveL 1024 to (-155.36, 322.12, -10) mm, rotated rx -180 ry 0 rz 0.01 deg; joints [40.321, -43.007, 97.443, -134.06, 64.246, 156.673]
  MoveL 1025 to (-155.9, 322.85, -10) mm, rotated rx -180 ry 0 rz 0.01 deg; joints [40.328, -42.965, 97.356, -134.037, 64.217, 156.634]
  MoveL 1026 to (-156.25, 323.26, -10) mm, rotated rx -180 ry 0 rz 0.01 deg; joints [40.331, -42.94, 97.303, -134.024, 64.199, 156.61]
  MoveL 1027 to (-163.73, 330.51, -10) mm, rotated rx 180 ry 0 rz 0.01 deg; joints [40.356, -42.448, 96.273, -133.81, 63.836, 156.168]
  MoveL 1028 to (-163.85, 330.62, -10) mm, rotated rx 180 ry 0 rz 0.01 deg; joints [40.357, -42.44, 96.257, -133.807, 63.831, 156.161]
  MoveL 1029 to (-165.86, 332.4, -10) mm, rotated rx 180 ry 0 rz 0.01 deg; joints [40.358, -42.312, 95.989, -133.755, 63.735, 156.048]
  MoveL 1030 to (-166.59, 332.89, -10) mm, rotated rx -180 ry 0 rz 0.01 deg; joints [40.355, -42.27, 95.902, -133.742, 63.702, 156.012]
  MoveL 1031 to (-177.84, 338.49, -10) mm, rotated rx -180 ry 0 rz 0.01 deg; joints [40.246, -41.682, 94.675, -133.621, 63.214, 155.547]
  MoveL 1032 to (-178.21, 338.64, -10) mm, rotated rx 180 ry 0 rz 0.01 deg; joints [40.242, -41.663, 94.636, -133.618, 63.199, 155.533]
  MoveL 1033 to (-178.93, 338.9, -10) mm, rotated rx -180 ry 0 rz 0.01 deg; joints [40.232, -41.628, 94.563, -133.614, 63.168, 155.506]
  MoveL 1034 to (-179.55, 339.06, -10) mm, rotated rx -180 ry 0 rz 0.01 deg; joints [40.222, -41.6, 94.506, -133.613, 63.143, 155.487]
  MoveL 1035 to (-180.49, 339.2, -10) mm, rotated rx 180 ry 0 rz 0.01 deg; joints [40.205, -41.56, 94.423, -133.616, 63.106, 155.46]
  MoveL 1036 to (4.87, 339.21, -10) mm, rotated rx 180 ry 0 rz 0.01 deg; joints [44.905, -47.839, 107.486, -131.124, 69.607, 159.005]
